//節流
ErrorSingle[1](
	bAutoStatus:=AutoStatus,
	bResetPB:=PB_Reset OR HMIPB_PB_Reset,
	bBackLS:=LS_S8_THBack,
	bOutLS:=LS_S8_THOut,
	bSOL:=SOL_S8_TH,
	bErrorStatus_Back=>Error_LS_S8_THBack,
	bErrorStatus_Out=>Error_LS_S8_THOut);
//換卡子
ErrorSingle[2](
	bAutoStatus:=AutoStatus,
	bResetPB:=PB_Reset OR HMIPB_PB_Reset,
	bBackLS:=LS_S8_FixBack,
	bOutLS:=LS_S8_FixOut,
	bSOL:=SOL_S8_Fix,
	bErrorStatus_Back=>Error_LS_S8_FixBack,
	bErrorStatus_Out=>Error_LS_S8_FixOut);
ErrorSingle[3](
	bAutoStatus:=AutoStatus,
	bResetPB:=PB_Reset OR HMIPB_PB_Reset,
	bBackLS:=LS_S8_FixMoveBack,
	bOutLS:=LS_S8_FixMoveOut,
	bSOL:=SOL_S8_FixMove,
	bErrorStatus_Back=>Error_LS_S8_FixMoveBack,
	bErrorStatus_Out=>Error_LS_S8_FixMoveOut);
ErrorSingle[4](
	bAutoStatus:=AutoStatus,
	bResetPB:=PB_Reset OR HMIPB_PB_Reset,
	bBackLS:=LS_S8_TurnBack,
	bOutLS:=LS_S8_TurnOut,
	bSOL:=SOL_S8_Turn,
	bErrorStatus_Back=>Error_LS_S8_TurnBack,
	bErrorStatus_Out=>Error_LS_S8_TurnOut);
ErrorSingle[5](
	bAutoStatus:=AutoStatus,
	bResetPB:=PB_Reset OR HMIPB_PB_Reset,
	bBackLS:=LS_S8_ClipBack,
	bOutLS:=LS_S8_ClipOut,
	bSOL:=SOL_S8_Clip,
	bErrorStatus_Back=>Error_LS_S8_ClipBack,
	bErrorStatus_Out=>Error_LS_S8_ClipOut);
//異常
ErrorStatus[8]:=
Error_LS_S8_MoveBack OR
Error_LS_S8_MoveBack OR
Error_LS_S8_UpDownBack OR
Error_LS_S8_UpDownOut OR
Error_SNR_S8_VacuumF OR
Error_SNR_S8_VacuumR OR
Error_OMRON_FQ2_Error;

ErrorStatus_TH[8]:=
Error_LS_S8_THBack OR
Error_LS_S8_THOut;

ErrorStatus_S8_Fix:=
Error_LS_S8_FixBack OR
Error_LS_S8_FixOut OR
Error_LS_S8_FixMoveBack OR
Error_LS_S8_FixMoveOut OR
Error_LS_S8_TurnBack OR
Error_LS_S8_TurnOut OR
Error_LS_S8_ClipBack OR
Error_LS_S8_ClipOut;
//RESET
IF PB_Reset OR HMIPB_PB_Reset THEN
	Error_SNR_S8_VacuumF:=FALSE;
	Error_SNR_S8_VacuumR:=FALSE;
	Error_OMRON_FQ2_Error:=FALSE;
END_IF;
END_PROGRAM

PROGRAM prError_S10
VAR
    ErrorDouble : ARRAY[0..9] of fbErrorDouble;
    ErrorSingle : ARRAY[0..9] of fbErrorSingle;
END_VAR
VAR_EXTERNAL
    AutoStatus : BOOL;
    PB_Reset : BOOL;
    HMIPB_PB_Reset : BOOL;
    LS_S10_MoveBack : BOOL;
    LS_S10_MoveOut : BOOL;
    SOL_S10_MoveBack : BOOL;
    SOL_S10_MoveOut : BOOL;
    Error_LS_S10_MoveBack : BOOL;
    Error_LS_S10_MoveOut : BOOL;
    LS_S10_UpDownBack : BOOL;
    LS_S10_UpDownOut : BOOL;
    SOL_S10_UpDown : BOOL;
    Error_LS_S10_UpDownBack : BOOL;
    Error_LS_S10_UpDownOut : BOOL;
    ErrorStatus : ARRAY[0..19] OF BOOL;
    ErrorStatus_TH : ARRAY[0..19] OF BOOL;
    LS_S10_THBack : BOOL;
    LS_S10_THOut : BOOL;
    SOL_S10_TH : BOOL;
    Error_LS_S10_THBack : BOOL;
    Error_LS_S10_THOut : BOOL;
    LS_S10_ClipFBack : BOOL;
    LS_S10_ClipFOut : BOOL;
    SOL_S10_ClipF : BOOL;
    Error_LS_S10_ClipFBack : BOOL;
    Error_LS_S10_ClipFOut : BOOL;
    LS_S10_ClipRBack : BOOL;
    LS_S10_ClipROut : BOOL;
    SOL_S10_ClipR : BOOL;
    Error_LS_S10_ClipRBack : BOOL;
    Error_LS_S10_ClipROut : BOOL;
END_VAR
//**********************************************************************************************************************
(*Station10*)
//**********************************************************************************************************************
ErrorDouble[0](
	bAutoStatus:=AutoStatus,
	bResetPB:=PB_Reset OR HMIPB_PB_Reset,
	bBackLS:=LS_S10_MoveBack,
	bOutLS:=LS_S10_MoveOut,
	bBackSOL:=SOL_S10_MoveBack,
	bOutSOL:=SOL_S10_MoveOut,
	bErrorStatus_Back=>Error_LS_S10_MoveBack,
	bErrorStatus_Out=>Error_LS_S10_MoveOut);

ErrorSingle[0](
	bAutoStatus:=AutoStatus,
	bResetPB:=PB_Reset OR HMIPB_PB_Reset,
	bBackLS:=LS_S10_UpDownBack,
	bOutLS:=LS_S10_UpDownOut,
	bSOL:=SOL_S10_UpDown,
	bErrorStatus_Back=>Error_LS_S10_UpDownBack,
	bErrorStatus_Out=>Error_LS_S10_UpDownOut);

ErrorSingle[1](
	bAutoStatus:=AutoStatus,
	bResetPB:=PB_Reset OR HMIPB_PB_Reset,
	bBackLS:=LS_S10_ClipFBack,
	bOutLS:=LS_S10_ClipFOut,
	bSOL:=SOL_S10_ClipF,
	bErrorStatus_Back=>Error_LS_S10_ClipFBack,
	bErrorStatus_Out=>Error_LS_S10_ClipFOut);

ErrorSingle[2](
	bAutoStatus:=AutoStatus,
	bResetPB:=PB_Reset OR HMIPB_PB_Reset,
	bBackLS:=LS_S10_ClipRBack,
	bOutLS:=LS_S10_ClipROut,
	bSOL:=SOL_S10_ClipR,
	bErrorStatus_Back=>Error_LS_S10_ClipRBack,
	bErrorStatus_Out=>Error_LS_S10_ClipROut);
//節流
ErrorSingle[3](
	bAutoStatus:=AutoStatus,
	bResetPB:=PB_Reset OR HMIPB_PB_Reset,
	bBackLS:=LS_S10_THBack,
	bOutLS:=LS_S10_THOut,
	bSOL:=SOL_S10_TH,
	bErrorStatus_Back=>Error_LS_S10_THBack,
	bErrorStatus_Out=>Error_LS_S10_THOut);

//異常
ErrorStatus[10]:=
Error_LS_S10_MoveBack OR
Error_LS_S10_MoveBack OR
Error_LS_S10_UpDownBack OR
Error_LS_S10_UpDownOut OR
Error_LS_S10_ClipFBack OR
Error_LS_S10_ClipFOut OR
Error_LS_S10_ClipRBack OR
Error_LS_S10_ClipROut;

ErrorStatus_TH[10]:=
Error_LS_S10_THBack OR
Error_LS_S10_THOut;
END_PROGRAM

PROGRAM prError_S11
VAR
    ErrorSingle : ARRAY[0..1] of fbErrorSingle;
END_VAR
VAR_EXTERNAL
    AutoStatus : BOOL;
    PB_Reset : BOOL;
    HMIPB_PB_Reset : BOOL;
    LS_S11_UpDownBack : BOOL;
    LS_S11_UpDownOut : BOOL;
    SOL_S11_UpDown : BOOL;
    Error_LS_S11_UpDownBack : BOOL;
    Error_LS_S11_UpDownOut : BOOL;
    ErrorStatus : ARRAY[0..19] OF BOOL;
END_VAR
//**********************************************************************************************************************
(*Station11*)
//**********************************************************************************************************************
ErrorSingle[0](
	bAutoStatus:=AutoStatus,
	bResetPB:=PB_Reset OR HMIPB_PB_Reset,
	bBackLS:=LS_S11_UpDownBack,
	bOutLS:=LS_S11_UpDownOut,
	bSOL:=SOL_S11_UpDown,
	bErrorStatus_Back=>Error_LS_S11_UpDownBack,
	bErrorStatus_Out=>Error_LS_S11_UpDownOut);

ErrorStatus[11]:=
Error_LS_S11_UpDownBack OR
Error_LS_S11_UpDownOut;
END_PROGRAM

PROGRAM prError_S13
VAR
    ErrorSingle : ARRAY[0..1] of fbErrorSingle;
END_VAR
VAR_EXTERNAL
    AutoStatus : BOOL;
    PB_Reset : BOOL;
    HMIPB_PB_Reset : BOOL;
    LS_S13_UpDownBack : BOOL;
    LS_S13_UpDownOut : BOOL;
    SOL_S13_UpDown : BOOL;
    Error_LS_S13_UpDownBack : BOOL;
    Error_LS_S13_UpDownOut : BOOL;
    ErrorStatus : ARRAY[0..19] OF BOOL;
END_VAR
//**********************************************************************************************************************
(*Station13*)
//**********************************************************************************************************************
ErrorSingle[0](
	bAutoStatus:=AutoStatus,
	bResetPB:=PB_Reset OR HMIPB_PB_Reset,
	bBackLS:=LS_S13_UpDownBack,
	bOutLS:=LS_S13_UpDownOut,
	bSOL:=SOL_S13_UpDown,
	bErrorStatus_Back=>Error_LS_S13_UpDownBack,
	bErrorStatus_Out=>Error_LS_S13_UpDownOut);

ErrorStatus[13]:=
Error_LS_S13_UpDownBack OR
Error_LS_S13_UpDownOut;
END_PROGRAM

PROGRAM prError_S15
VAR
    ErrorSingle : ARRAY[0..1] of fbErrorSingle;
END_VAR
VAR_EXTERNAL
    AutoStatus : BOOL;
    PB_Reset : BOOL;
    HMIPB_PB_Reset : BOOL;
    LS_S15_UpDownBack : BOOL;
    LS_S15_UpDownOut : BOOL;
    SOL_S15_UpDown : BOOL;
    Error_LS_S15_UpDownBack : BOOL;
    Error_LS_S15_UpDownOut : BOOL;
    ErrorStatus : ARRAY[0..19] OF BOOL;
END_VAR
//**********************************************************************************************************************
(*Station15*)
//**********************************************************************************************************************
ErrorSingle[0](
	bAutoStatus:=AutoStatus,
	bResetPB:=PB_Reset OR HMIPB_PB_Reset,
	bBackLS:=LS_S15_UpDownBack,
	bOutLS:=LS_S15_UpDownOut,
	bSOL:=SOL_S15_UpDown,
	bErrorStatus_Back=>Error_LS_S15_UpDownBack,
	bErrorStatus_Out=>Error_LS_S15_UpDownOut);

ErrorStatus[15]:=
Error_LS_S15_UpDownBack OR
Error_LS_S15_UpDownOut;
END_PROGRAM

PROGRAM prStation1
VAR
    AutoFlow : INT;
    Rtrig_test : R_TRIG;
    TON_CT : TON;
END_VAR
VAR_EXTERNAL
    IndexData : ARRAY[0..19] OF stIndexData;
    DisablePB : ARRAY[0..19] OF BOOL;
    TestPB : ARRAY[0..19] OF BOOL;
    SystemReadyStatus : BOOL;
    AutoStatus : BOOL;
    ErrorStatus : ARRAY[0..19] OF BOOL;
    Error_PB_EStop : BOOL;
    YAMAHA_Load_Start : BOOL;
    MachineRunStatus : BOOL;
    YAMAHA_Load_Finish : BOOL;
    CycleTime : ARRAY[0..19] OF REAL;
    BatchIndexCount : DINT;
    HMIPB_YAMAHA_Load_Start : BOOL;
    HMIPB_OMRON_FQ2_Trig : BOOL;
    Error_LS_Door : BOOL;
    StepMode : BOOL;
END_VAR
(*
程序名稱:第1站上料流程
作者:蔡相偉
版本,日期,版本資訊:
1.0.0		2017/11/21		初始版本
PowerOn=0
Idle=1
上料開始=2
上料完成=3
*)
//本站狀態判斷
IF IndexData[1].OKFlag[1]
	OR IndexData[1].NGFlag[1] THEN
	IndexData[1].FinishFlag[1]:=TRUE;
END_IF;
(*
//前站狀態判斷
IF NOT(IndexData[10].FinishFlag[9]
	AND IndexData[10].OKFlag[9]
	AND NOT(IndexData[10].NGFlag[9])) THEN
	IndexData[10].NGFlag[10]:=TRUE;
END_IF;
*)
//本站關閉判斷
IF DisablePB[1] AND NOT(IndexData[1].FinishFlag[1]) THEN
	IndexData[1].NGFlag[1]:=TRUE;
END_IF;
//異常放棄
IF (ErrorStatus[1] OR Error_PB_EStop) AND NOT(IndexData[1].FinishFlag[1]) THEN
	IndexData[1].NGFlag[1]:=TRUE;
END_IF;

Rtrig_test(CLK:=TestPB[1]);
//PowerOn=0
IF NOT(SystemReadyStatus AND AutoStatus AND NOT(ErrorStatus[1]) AND NOT(Error_PB_EStop)) THEN
	Autoflow:=0;
END_IF;

//Idle=1
IF AutoFlow=0 AND SystemReadyStatus AND AutoStatus AND NOT(ErrorStatus[1]) AND NOT(Error_PB_EStop) THEN
	AutoFlow:=1;
END_IF;

IF AutoFlow=3 AND NOT(YAMAHA_Load_Start) AND IndexData[1].FinishFlag[1] THEN
	AutoFlow:=1;
END_IF;

//上料開始=2
IF Autoflow=1
	AND AutoStatus
	AND NOT(DisablePB[1])
	AND (MachineRunStatus AND NOT(IndexData[1].FinishFlag[1]) OR Rtrig_test.Q) THEN
	Autoflow:=2;
END_IF;
IF AutoFlow=2 THEN
	HMIPB_YAMAHA_Load_Start:=TRUE;
END_IF;
IF YAMAHA_Load_Finish OR ErrorStatus[1] OR Error_LS_Door THEN
	HMIPB_YAMAHA_Load_Start:=FALSE;
END_IF;

//上料完成=3
IF AutoFlow=2 AND (YAMAHA_Load_Finish) THEN
	BatchIndexCount:=BatchIndexCount+1;
	AutoFlow:=3;
END_IF;
IF AutoFlow=3 THEN
	IndexData[1].OKFlag[1]:=TRUE;
END_IF;
//IndexCount
(*IF BatchIndexCount<0 THEN
	BatchIndexCount:=0;
END_IF;*)
//*************************************************************************
//Cycle Time
//*************************************************************************
TON_CT(In:=AutoFlow>1, PT:=t#500s);
IF AutoFlow>1 THEN
CycleTime[1]:=LINT_TO_REAL(TimeToNanoSec( TON_CT.ET))/1000000000.0;
END_IF;
END_PROGRAM

PROGRAM prStation1_Robot
VAR
    R_TRIG1 : R_TRIG;
    R_TRIG2 : R_TRIG;
    R_TRIG3 : R_TRIG;
END_VAR
VAR_EXTERNAL
    HMIPB_YAMAHA_Unload_OKStart : BOOL;
    YAMAHA_Unload_OKStart : BOOL;
    YAMAHA_Unload_NGStart : BOOL;
    HMIPB_YAMAHA_Unload_NGStart : BOOL;
    YAMAHA_Load_Start : BOOL;
    HMIPB_YAMAHA_Load_Start : BOOL;
    YAMAHA_UnLoad_Ready : BOOL;
    HMIPB_YAMAHA_UnLoad_Ready : BOOL;
    HMIPB_YAMAHA_Load_Ready : BOOL;
    YAMAHA_Load_Ready : BOOL;
    HMIPB_YAMAHA_Unload_ChangePanelStart : BOOL;
    YAMAHA_Unload_ChangePanelStart : BOOL;
    HMIPB_YAMAHA_Load_ChangePanelStart : BOOL;
    YAMAHA_Load_ChangePanelStart : BOOL;
    HMIPB_YAMAHA_ORG : BOOL;
    YAMAHA_ORG : BOOL;
    HMIPB_YAMAHA_S_Enable : BOOL;
    YAMAHA_S_Enable : BOOL;
    HMIPB_YAMAHA_S_Control : BOOL;
    YAMAHA_S_Control : BOOL;
    HMIPB_YAMAHA_S_Stop : BOOL;
    YAMAHA_S_Stop : BOOL;
    HMIPB_YAMAHA_S_AutoRun : BOOL;
    YAMAHA_S_AutoRun : BOOL;
    HMIPB_YAMAHA_S_INCHome : BOOL;
    YAMAHA_S_INCHome : BOOL;
    HMIPB_YAMAHA_S_ProgramReset : BOOL;
    YAMAHA_S_ProgramReset : BOOL;
    HMIPB_YAMAHA_S_AlarmReset : BOOL;
    YAMAHA_S_AlarmReset : BOOL;
    HMIPB_YAMAHA_S_ABSHome : BOOL;
    YAMAHA_S_ABSHome : BOOL;
    PB_EStop : BOOL;
    SNR_S1_Door1 : BOOL;
    SNR_S1_Door2 : BOOL;
    SNR_S1_Door3 : BOOL;
    SNR_S1_Door4 : BOOL;
    SystemReadyStatus : BOOL;
    YAMAHA_S_State_CPUOK : BOOL;
    YAMAHA_S_State_Enable : BOOL;
    Error_PB_EStop : BOOL;
    Error_LS_Door : BOOL;
    YAMAHA_S_State_Homed : BOOL;
    YAMAHA_S_State_ProgramReset : BOOL;
    YAMAHA_S_State_RobotProgramRun : BOOL;
END_VAR
//Define
YAMAHA_Unload_OKStart:=HMIPB_YAMAHA_Unload_OKStart;
YAMAHA_Unload_NGStart:=HMIPB_YAMAHA_Unload_NGStart;
YAMAHA_Load_Start:=HMIPB_YAMAHA_Load_Start;
//YAMAHA_UnLoad_Ready:=HMIPB_YAMAHA_UnLoad_Ready;
//YAMAHA_Load_Ready:=HMIPB_YAMAHA_Load_Ready;
YAMAHA_S_Control:=HMIPB_YAMAHA_S_Control;
YAMAHA_S_AutoRun:=HMIPB_YAMAHA_S_AutoRun;
YAMAHA_S_INCHome:=HMIPB_YAMAHA_S_INCHome;
YAMAHA_S_ProgramReset:=HMIPB_YAMAHA_S_ProgramReset;
YAMAHA_S_AlarmReset:=HMIPB_YAMAHA_S_AlarmReset;
YAMAHA_S_ABSHome:=HMIPB_YAMAHA_S_ABSHome;

//********************************************************************************************************
//ROBOT伺服ON流程
//********************************************************************************************************
R_TRIG1(Clk:=(SystemReadyStatus AND YAMAHA_S_State_CPUOK) OR HMIPB_YAMAHA_S_Enable);
IF R_TRIG1.Q THEN
	YAMAHA_S_Enable:=TRUE;
END_IF;
IF YAMAHA_S_State_Enable THEN
	YAMAHA_S_Enable:=FALSE;
END_IF;
//********************************************************************************************************
//STOP ON
//********************************************************************************************************
YAMAHA_S_Stop:=
HMIPB_YAMAHA_S_Stop AND
NOT(Error_PB_EStop) AND
NOT(Error_LS_Door);
//********************************************************************************************************
//程序復位和執行
//********************************************************************************************************
R_TRIG2(Clk:=YAMAHA_S_State_Homed AND YAMAHA_S_State_Enable AND YAMAHA_S_Stop AND HMIPB_YAMAHA_S_ProgramReset);
R_TRIG3(Clk:=YAMAHA_S_State_Homed AND YAMAHA_S_State_Enable AND YAMAHA_S_Stop AND YAMAHA_S_State_ProgramReset AND HMIPB_YAMAHA_S_AutoRun);
IF R_TRIG2.Q THEN
	YAMAHA_S_ProgramReset:=TRUE;
END_IF;
IF YAMAHA_S_State_ProgramReset THEN
	HMIPB_YAMAHA_S_ProgramReset:=FALSE;
END_IF;
IF R_TRIG3.Q THEN
	YAMAHA_S_AutoRun:=TRUE;
END_IF;
IF YAMAHA_S_State_RobotProgramRun AND NOT(YAMAHA_S_State_ProgramReset) THEN
	YAMAHA_S_AutoRun:=FALSE;
	HMIPB_YAMAHA_S_AutoRun:=FALSE;
END_IF;
END_PROGRAM

PROGRAM prStation1_PanelLoad
VAR
    Autoflow : INT;
    Initflow : INT;
    interlockback : ARRAY[0..2] OF BOOL;
    interlockout : ARRAY[0..2] OF BOOL;
    solStatus : ARRAY[0..2] OF BOOL;
    R_TRIG_1 : ARRAY[0..2] OF R_TRIG;
    F_TRIG_1 : F_TRIG;
    ErrorLS : BOOL;
    StartFlag : BOOL;
    TON_1 : TON;
    TON_2 : TON;
    TON_3 : TON;
    Rtrig_test : R_TRIG;
END_VAR
VAR_EXTERNAL
    HMIPB_SOL_S1_Load_PanelUpDown1Back : BOOL;
    SOL_S1_Load_PanelUpDown1Back : BOOL;
    SOL_S1_Load_PanelUpDown1Out : BOOL;
    LS_S1_Load_PanelUpDown1Back : BOOL;
    HMIPB_SOL_S1_Load_PanelUpDown1Out : BOOL;
    AutoStatus : BOOL;
    LS_S1_Load_PanelUpDown1Out : BOOL;
    HMIPB_SOL_S1_Load_PanelUpDown2Back : BOOL;
    SOL_S1_Load_PanelUpDown2Back : BOOL;
    SOL_S1_Load_PanelUpDown2Out : BOOL;
    LS_S1_Load_PanelUpDown2Back : BOOL;
    HMIPB_SOL_S1_Load_PanelUpDown2Out : BOOL;
    LS_S1_Load_PanelUpDown2Out : BOOL;
    HMIPB_SOL_S1_Load_PanelClip : BOOL;
    SOL_S1_Load_PanelClip : BOOL;
    SystemReadyStatus : BOOL;
    ErrorStatus : ARRAY[0..19] OF BOOL;
    Error_PB_EStop : BOOL;
    SNR_S1_Load_PanelFeed : BOOL;
    LS_S1_Load_PanelClip1Out : BOOL;
    LS_S1_Load_PanelClip2Out : BOOL;
    LS_S1_Load_PanelClip2Back : BOOL;
    LS_S1_Load_PanelClip1Back : BOOL;
    RY_S1_Load_VariableSpeedMotor : BOOL;
    Error_LS_S1_Load_PanelUpDown1Back : BOOL;
    Error_LS_S1_Load_PanelUpDown1Out : BOOL;
    Error_LS_S1_Load_PanelUpDown2Back : BOOL;
    Error_LS_S1_Load_PanelUpDown2Out : BOOL;
    Error_LS_S1_Load_PanelClip1Back : BOOL;
    Error_LS_S1_Load_PanelClip1Out : BOOL;
    Error_LS_S1_Load_PanelClip2Back : BOOL;
    Error_LS_S1_Load_PanelClip2Out : BOOL;
    ErrorStatus_S1_Load : BOOL;
    Error_SNR_S1_Load_PanelFeed : BOOL;
    PB_Reset : BOOL;
    HMIPB_PB_Reset : BOOL;
    StepMode : BOOL;
    Manual2AutoFlag : BOOL;
END_VAR
(*
程序名稱: Panel LOAD程序
作者:蔡相偉
版本,日期,版本資訊:
1.0.0		2017/11/16		初始版本

PowerOn=0
Idle=1
Panel出盤程序開始=10
第1段,第2段出=2
夾持出=3
第2段回=4
夾持回=5
第1段回=6
第1段到回=7
*)
//***************************************************************************************************************
//Define
ErrorLS:=ErrorStatus_S1_Load;
StartFlag:=TON_1.Q;
TON_1(In:=NOT(SNR_S1_Load_PanelFeed) AND NOT(RY_S1_Load_VariableSpeedMotor), PT:=t#5s);
//PowerOn=0
IF NOT(SystemReadyStatus AND NOT(ErrorLS) AND  NOT(Error_PB_Estop) AND AutoStatus) THEN
	Autoflow:=0;
END_IF;

//Idle=1
IF AutoFlow=0 AND SystemReadyStatus AND NOT(ErrorLS) AND  NOT(Error_PB_Estop) AND AutoStatus THEN
	AutoFlow:=1;
END_IF;

IF Autoflow=7 AND (Error_SNR_S1_Load_PanelFeed OR SNR_S1_Load_PanelFeed) THEN
	Autoflow:=1;
END_IF;

//第1段,第2段出=2
IF Autoflow=1 AND NOT(Error_SNR_S1_Load_PanelFeed) AND StartFlag THEN
	Autoflow:=2;
END_IF;

//承盤夾持出=3
IF Autoflow=2 AND LS_S1_Load_PanelUpDown1Out AND LS_S1_Load_PanelUpDown2Out AND (Rtrig_test.Q OR NOT(StepMode)) THEN
	Autoflow:=3;
END_IF;
TON_2(In:= Autoflow=3 AND LS_S1_Load_PanelClip1Out AND LS_S1_Load_PanelClip2Out , PT:=t#300ms);

//第2段回=4
IF Autoflow=3 AND TON_2.Q AND (Rtrig_test.Q OR NOT(StepMode)) THEN
	Autoflow:=4;
END_IF;
TON_3(In:=Autoflow=4 AND LS_S1_Load_PanelUpDown2Back, PT:=t#300ms);

//承盤夾持回=5
IF Autoflow=4 AND TON_3.Q AND (Rtrig_test.Q OR NOT(StepMode)) THEN
	Autoflow:=5;
END_IF;

//第1段回=6
IF Autoflow=5 AND  LS_S1_Load_PanelClip1Back AND LS_S1_Load_PanelClip2Back AND (Rtrig_test.Q OR NOT(StepMode)) THEN
	Autoflow:=6;
END_IF;

//第1段到回=7
IF Autoflow=6 AND  LS_S1_Load_PanelUpDown1Back AND (Rtrig_test.Q OR NOT(StepMode)) THEN
	Autoflow:=7;
END_IF;
IF Autoflow=7 AND NOT(SNR_S1_Load_PanelFeed) THEN
	Error_SNR_S1_Load_PanelFeed:=TRUE;
END_IF;

//***************************************************************************************************************
//下夾板出盤下降第1段回電磁閥
interlockback[0]:=TRUE;
IF ((HMIPB_SOL_S1_Load_PanelUpDown1Back AND NOT(AutoStatus)) OR Autoflow=6 OR Initflow=3) AND interlockback[0] THEN
	SOL_S1_Load_PanelUpDown1Back:=TRUE;
	SOL_S1_Load_PanelUpDown1Out:=FALSE;
END_IF;
IF LS_S1_Load_PanelUpDown1Back THEN
	SOL_S1_Load_PanelUpDown1Back:=FALSE;
END_IF;

//下夾板出盤下降第1段出電磁閥
interlockout[0]:=TRUE;
IF ((HMIPB_SOL_S1_Load_PanelUpDown1Out AND NOT(AutoStatus)) OR Autoflow=2) AND interlockout[0] THEN
	SOL_S1_Load_PanelUpDown1Back:=FALSE;
	SOL_S1_Load_PanelUpDown1Out:=TRUE;
END_IF;
IF LS_S1_Load_PanelUpDown1Out THEN
	SOL_S1_Load_PanelUpDown1Out:=FALSE;
END_IF;
//***************************************************************************************************************
//下夾板出盤下降第2段回電磁閥
interlockback[1]:=TRUE;
IF ((HMIPB_SOL_S1_Load_PanelUpDown2Back AND NOT(AutoStatus)) OR Autoflow=4 OR Initflow=3) AND interlockback[1] THEN
	SOL_S1_Load_PanelUpDown2Back:=TRUE;
	SOL_S1_Load_PanelUpDown2Out:=FALSE;
END_IF;
IF LS_S1_Load_PanelUpDown2Back THEN
	SOL_S1_Load_PanelUpDown2Back:=FALSE;
END_IF;

//下夾板出盤下降第2段出電磁閥
interlockout[1]:=LS_S1_Load_PanelUpDown1Out AND NOT(SNR_S1_Load_PanelFeed);
IF ((HMIPB_SOL_S1_Load_PanelUpDown2Out AND NOT(AutoStatus)) OR Autoflow=2) AND interlockout[1] THEN
	SOL_S1_Load_PanelUpDown2Back:=FALSE;
	SOL_S1_Load_PanelUpDown2Out:=TRUE;
END_IF;
IF LS_S1_Load_PanelUpDown2Out THEN
	SOL_S1_Load_PanelUpDown2Out:=FALSE;
END_IF;
//***************************************************************************************************************
(*下夾板出盤承載電磁閥*)
R_TRIG_1[2](CLK:=HMIPB_SOL_S1_Load_PanelClip AND NOT(AutoStatus));
interlockback[2]:=TRUE;
interlockout[2]:=LS_S1_Load_PanelUpDown1Out;
(*SET*)
IF ((R_TRIG_1[2].Q AND NOT(solStatus[2])) OR Autoflow=3) AND interlockout[2] THEN
	SOL_S1_Load_PanelClip:=TRUE;
END_IF;
(*RESET*)
IF ((R_TRIG_1[2].Q AND (solStatus[2])) OR Autoflow=5 OR Initflow=2) AND interlockback[2] THEN
	SOL_S1_Load_PanelClip:=FALSE;
END_IF;
(*STATUS*)
solStatus[2]:=SOL_S1_Load_PanelClip;

//***************************************************************************************************************
(*
程序名稱: Panel LOAD RESET程序
作者:蔡相偉
版本,日期,版本資訊:
1.0.0		2017/11/16		初始版本

PowerOn=0
Idle=1
夾持回=2
第1段回,第2段回=3
*)
//***************************************************************************************************************
//PowerOn=0
IF NOT(SystemReadyStatus) THEN
	Initflow:=0;
END_IF;

//Idle=1
IF Initflow=0 AND SystemReadyStatus THEN
	Initflow:=1;
END_IF;

IF Initflow=3 AND LS_S1_Load_PanelUpDown1Back AND LS_S1_Load_PanelUpDown2Back THEN
	Initflow:=1;
END_IF;

F_TRIG_1(Clk:=ErrorLS OR Error_PB_Estop);
//夾持回=2
IF Initflow=1 AND (F_TRIG_1.Q OR Manual2AutoFlag) THEN
	Initflow:=2;
END_IF;

//第1段回,第2段回=3
IF Initflow=2 AND LS_S1_Load_PanelClip1Back AND LS_S1_Load_PanelClip2Back THEN
	Initflow:=3;
END_IF;
END_PROGRAM

PROGRAM prStation1_FeedPanelLoad
VAR
    Autoflow : INT;
    interlockback : ARRAY[0..3] OF BOOL;
    interlockout : ARRAY[0..3] OF BOOL;
    solStatus : ARRAY[0..3] OF BOOL;
    R_TRIG_1 : ARRAY[0..3] OF R_TRIG;
    ErrorLS : BOOL;
    StartFlag : BOOL;
    TON_1 : TON;
    TON_2 : TON;
    TON_3 : TON;
    TON_4 : TON;
    TON_5 : TON;
    TON_6 : TON;
    F_TRIG_1 : F_TRIG;
    centermotorStartflag : BOOL;
    Rtrig_test : R_TRIG;
    Initflow : INT;
END_VAR
VAR_EXTERNAL
    HMIPB_SOL_S1_Load_PanelUpDown1Back : BOOL;
    SOL_S1_Load_PanelUpDown1Back : BOOL;
    SOL_S1_Load_PanelUpDown1Out : BOOL;
    LS_S1_Load_PanelUpDown1Back : BOOL;
    HMIPB_SOL_S1_Load_PanelUpDown1Out : BOOL;
    AutoStatus : BOOL;
    LS_S1_Load_PanelUpDown1Out : BOOL;
    HMIPB_SOL_S1_Load_PanelUpDown2Back : BOOL;
    SOL_S1_Load_PanelUpDown2Back : BOOL;
    SOL_S1_Load_PanelUpDown2Out : BOOL;
    LS_S1_Load_PanelUpDown2Back : BOOL;
    HMIPB_SOL_S1_Load_PanelUpDown2Out : BOOL;
    LS_S1_Load_PanelUpDown2Out : BOOL;
    HMIPB_SOL_S1_Load_PanelClip : BOOL;
    SOL_S1_Load_PanelClip : BOOL;
    HMIPB_SOL_S1_Load_FixClip : BOOL;
    SOL_S1_Load_FixClip : BOOL;
    HMIPB_SOL_S1_Load_ConveyorClip : BOOL;
    SOL_S1_Load_ConveyorClip : BOOL;
    HMIPB_SOL_S1_Load_UpDown : BOOL;
    SOL_S1_Load_UpDown : BOOL;
    HMIPB_RY_S1_Load_VariableSpeedMotor : BOOL;
    RY_S1_Load_VariableSpeedMotor : BOOL;
    RY_S1_Load_FixSpeedMotor : BOOL;
    HMIPB_RY_S1_Load_FixSpeedMotor : BOOL;
    SNR_S1_Load_PanelFeed : BOOL;
    SNR_S1_Load_PanelClip : BOOL;
    SystemReadyStatus : BOOL;
    ErrorStatus : ARRAY[0..19] OF BOOL;
    ErrorStatus_TH : ARRAY[0..19] OF BOOL;
    RY_S1_Center_VariableSpeedMotor : BOOL;
    HMIPB_RY_S1_Center_VariableSpeedMotor : BOOL;
    Error_PB_EStop : BOOL;
    ErrorStatus_S1_FeedPanelLoad : BOOL;
    HMIPB_SOL_S1_Load_AlignmentClip : BOOL;
    SOL_S1_Load_AlignmentClip : BOOL;
    YAMAHA_Load_ChangePanelStart : BOOL;
    HMIPB_YAMAHA_Load_ChangePanelStart : BOOL;
    SNR_AirSource : BOOL;
    SNR_S1_Load_Feed : BOOL;
    SNR_S1_UnLoad_Feed : BOOL;
    LS_S1_Load_FixClipOut : BOOL;
    LS_S1_Load_AlignmentClipOut : BOOL;
    HMIPB_YAMAHA_Unload_ChangePanelStart : BOOL;
    LS_S1_Load_UpDownOut : BOOL;
    LS_S1_Load_ConveyorClip1Out : BOOL;
    LS_S1_Load_ConveyorClip2Out : BOOL;
    LS_S10_ClipFBack : BOOL;
    LS_S1_Load_UpDownBack : BOOL;
    LS_S1_Load_ConveyorClip1Back : BOOL;
    LS_S1_Load_ConveyorClip2Back : BOOL;
    LS_S1_Load_FixClipBack : BOOL;
    LS_S1_Load_AlignmentClipBack : BOOL;
    YAMAHA_Load_Ready : BOOL;
    YAMAHA_Load_Finish : BOOL;
    YAMAHA_Load_Start : BOOL;
    YAMAHA_Unload_ChangePanelStart : BOOL;
    LS_S1_UnLoad_UpDownBack : BOOL;
    SOL_S1_UnLoad_UpDown : BOOL;
    StepMode : BOOL;
    LS_S1_UnLoad_PanelUpDown1Back : BOOL;
    LS_S1_UnLoad_PanelUpDown2Back : BOOL;
    Manual2AutoFlag : BOOL;
    LS_S1_UnLoad_PanelClip1Back : BOOL;
    LS_S1_UnLoad_PanelClip2Back : BOOL;
END_VAR
(*
程序名稱: 出盤程序
作者:蔡相偉
版本,日期,版本資訊:
1.0.0		2017/11/16		初始版本

PowerOn=0--->
Idle=1--->
換盤程序開始=2|--->工件取放處有盤=10--->固定,活動夾持出=11--->上下出=12--->軌道夾持出=13--->上下回=14--->軌道夾持回=15--->20
						  |--->工件取放處無盤=20--->軌道夾持回=21--->固定,活動夾持出=22--->馬達ON=23--->馬達運行中=24--->盤到位,馬達停止=25--->固定邊夾持回=26--->活動邊夾持回=27--->換盤完成=28--->1
*)
(*
Error Code
1:緊急停止
2:磁簧異常
*)
//***************************************************************************************************************
//Define
ErrorLS:=
ErrorStatus_S1_FeedPanelLoad;
//***************************************************************************************************************
//PowerOn=0
IF NOT(SystemReadyStatus AND NOT(ErrorLS) AND  NOT(Error_PB_Estop)) THEN
	Autoflow:=0;
END_IF;

//Idle=1
IF Autoflow=0 AND SystemReadyStatus AND NOT(ErrorLS) AND  NOT(Error_PB_Estop) THEN
	Autoflow:=1;
END_IF;

IF Autoflow=28 AND NOT(YAMAHA_Load_ChangePanelStart) AND NOT(HMIPB_YAMAHA_Load_ChangePanelStart) THEN
	Autoflow:=1;
END_IF;

TON_1(In:=Autoflow=1 AND NOT(SNR_S1_Load_PanelClip), PT:=t#1s);

IF Autoflow=1 AND TON_5.Q THEN		(*READY訊號*)
	YAMAHA_Load_Ready:=TRUE;
ELSE
	YAMAHA_Load_Ready:=FALSE;
END_IF;

//換盤程序開始=2
IF Autoflow=1 AND (YAMAHA_Load_ChangePanelStart OR HMIPB_YAMAHA_Load_ChangePanelStart OR TON_1.Q) AND SNR_S1_Load_PanelFeed THEN
	Autoflow:=2;
END_IF;

//工件取放處有盤=10
IF Autoflow=2 AND SNR_S1_Load_PanelClip THEN
	Autoflow:=10;
END_IF;

//固定,活動夾持出=11
IF Autoflow=10 THEN
	Autoflow:=11;
END_IF;
IF Autoflow=11 AND SNR_S1_Load_Feed THEN
	HMIPB_YAMAHA_Unload_ChangePanelStart:=TRUE;
END_IF;
TON_4(In:=Autoflow=11 AND NOT(SNR_S1_Load_Feed), PT:=t#1s);

//上下出=12
IF Autoflow=11 AND LS_S1_Load_FixClipOut AND LS_S1_Load_AlignmentClipOut AND TON_4.Q AND (Rtrig_test.Q OR NOT(StepMode)) THEN
	Autoflow:=12;
	HMIPB_YAMAHA_Unload_ChangePanelStart:=FALSE;
END_IF;

//軌道夾持出=13
IF Autoflow=12 AND LS_S1_Load_UpDownOut AND (Rtrig_test.Q OR NOT(StepMode)) THEN
	Autoflow:=13;
END_IF;

//上下回=14
IF Autoflow=13 AND LS_S1_Load_ConveyorClip1Out AND LS_S1_Load_ConveyorClip2Out AND (Rtrig_test.Q OR NOT(StepMode)) THEN
	Autoflow:=14;
END_IF;

//軌道夾持回=15
IF Autoflow=14 AND LS_S1_Load_UpDownBack AND (Rtrig_test.Q OR NOT(StepMode)) THEN
	Autoflow:=15;
END_IF;
//***************************************************************************************************************
//工件取放處無盤=20
IF Autoflow=2 AND NOT(SNR_S1_Load_PanelClip) THEN
	Autoflow:=20;
END_IF;

IF Autoflow=15 AND LS_S1_Load_ConveyorClip1Back AND LS_S1_Load_ConveyorClip2Back THEN
	Autoflow:=20;
END_IF;

//軌道夾持回=21
IF Autoflow=20 THEN
	Autoflow:=21;
END_IF;

//固定,活動夾持出=22
IF Autoflow=21 AND LS_S1_Load_ConveyorClip1Back AND LS_S1_Load_ConveyorClip2Back AND (Rtrig_test.Q OR NOT(StepMode)) THEN
	Autoflow:=22;
END_IF;

//馬達ON=23
IF Autoflow=22 AND LS_S1_Load_FixClipOut AND LS_S1_Load_AlignmentClipOut AND SNR_S1_Load_PanelFeed THEN
	Autoflow:=23;
END_IF;
IF Autoflow=23 THEN
	HMIPB_RY_S1_Load_FixSpeedMotor:=TRUE;
	HMIPB_RY_S1_Load_VariableSpeedMotor:=TRUE;
END_IF;

//馬達運行中=24
IF Autoflow=23 AND RY_S1_Load_FixSpeedMotor AND RY_S1_Load_VariableSpeedMotor THEN
	Autoflow:=24;
END_IF;


//盤到位,馬達停止=25
IF Autoflow=24 AND TON_5.Q THEN
	Autoflow:=25;
END_IF;


//固定邊夾持回=26
IF Autoflow=25 AND NOT(RY_S1_Load_FixSpeedMotor) AND (Rtrig_test.Q OR NOT(StepMode)) THEN
	Autoflow:=26;
END_IF;

//活動邊夾持回=27
IF Autoflow=26 AND LS_S1_Load_FixClipBack AND (Rtrig_test.Q OR NOT(StepMode)) THEN
	Autoflow:=27;
END_IF;
//換盤完成=28
IF Autoflow=27 AND LS_S1_Load_AlignmentClipBack THEN
	Autoflow:=28;
END_IF;

//***************************************************************************************************************
//下夾板出盤固定邊定位電磁閥
R_TRIG_1[0](CLK:=HMIPB_SOL_S1_Load_FixClip AND NOT(AutoStatus));
interlockback[0]:=TRUE;
interlockout[0]:=TRUE;
//SET
IF ((R_TRIG_1[0].Q AND NOT(solStatus[0])) OR Autoflow=11 OR Autoflow=22) AND interlockout[0] THEN
	SOL_S1_Load_FixClip:=TRUE;
END_IF;
//RESET
IF ((R_TRIG_1[0].Q AND (solStatus[0])) OR Autoflow=26 OR Initflow=26) AND interlockback[0] THEN
	SOL_S1_Load_FixClip:=FALSE;
END_IF;
//STATUS
solStatus[0]:=SOL_S1_Load_FixClip;
//***************************************************************************************************************
//下夾板出盤活動邊定位電磁閥
R_TRIG_1[1](CLK:=HMIPB_SOL_S1_Load_AlignmentClip AND NOT(AutoStatus));
interlockback[1]:=TRUE;
interlockout[1]:=TRUE;
//SET
IF ((R_TRIG_1[1].Q AND NOT(solStatus[1])) OR Autoflow=11 OR Autoflow=22) AND interlockout[1] THEN
	SOL_S1_Load_AlignmentClip:=TRUE;
END_IF;
//RESET
IF ((R_TRIG_1[1].Q AND (solStatus[1])) OR Autoflow=27 OR Initflow=27) AND interlockback[1] THEN
	SOL_S1_Load_AlignmentClip:=FALSE;
END_IF;
//STATUS
solStatus[1]:=SOL_S1_Load_AlignmentClip;
//***************************************************************************************************************
//下夾板出盤軌道開合電磁閥
R_TRIG_1[2](CLK:=HMIPB_SOL_S1_Load_ConveyorClip AND NOT(AutoStatus));
interlockback[2]:=TRUE;
interlockout[2]:=LS_S1_Load_UpDownOut AND SOL_S1_Load_UpDown;
//SET
IF ((R_TRIG_1[2].Q AND NOT(solStatus[2])) OR Autoflow=13) AND interlockout[2] THEN
	SOL_S1_Load_ConveyorClip:=TRUE;
END_IF;
//RESET
IF ((R_TRIG_1[2].Q AND (solStatus[2])) OR Autoflow=15 OR Autoflow=21 OR Initflow=21) AND interlockback[2] THEN
	SOL_S1_Load_ConveyorClip:=FALSE;
END_IF;
//STATUS
solStatus[2]:=SOL_S1_Load_ConveyorClip;
//***************************************************************************************************************
//下夾板出盤升降電磁閥
R_TRIG_1[3](CLK:=HMIPB_SOL_S1_Load_UpDown AND NOT(AutoStatus));
interlockback[3]:=TRUE;
interlockout[3]:=LS_S1_Load_AlignmentClipOut AND SOL_S1_Load_AlignmentClip AND LS_S1_Load_FixClipOut AND SOL_S1_Load_FixClip;
//RESET
IF ((R_TRIG_1[3].Q AND NOT(solStatus[3])) OR Autoflow=12) AND interlockout[3] THEN
	SOL_S1_Load_UpDown:=TRUE;
END_IF;
//RESET
IF ((R_TRIG_1[3].Q AND (solStatus[3])) OR Autoflow=14 OR Initflow=14) AND interlockback[3] THEN
	SOL_S1_Load_UpDown:=FALSE;
END_IF;
//STATUS
solStatus[3]:=SOL_S1_Load_UpDown;
//***************************************************************************************************************
//下夾板出盤調速馬達繼電器
//RESET
TON_6(In:=NOT(SNR_S1_Load_PanelFeed) AND LS_S1_Load_PanelUpDown1Back AND LS_S1_Load_PanelUpDown2Back, PT:=t#1s);
IF TON_6.Q THEN
	HMIPB_RY_S1_Load_VariableSpeedMotor:=FALSE;
END_IF;
//OUT
RY_S1_Load_VariableSpeedMotor:=HMIPB_RY_S1_Load_VariableSpeedMotor AND NOT(StepMode);
//***************************************************************************************************************
//下夾板出盤定速馬達繼電器
//RESET
TON_5(In:=SNR_S1_Load_PanelClip, PT:=t#1s);
IF TON_5.Q THEN
	HMIPB_RY_S1_Load_FixSpeedMotor:=FALSE;
END_IF;
//OUT
RY_S1_Load_FixSpeedMotor:=HMIPB_RY_S1_Load_FixSpeedMotor AND NOT(StepMode);
//***************************************************************************************************************
//下夾板下移載調速馬達繼電器
TON_2(In:=SNR_S1_Load_Feed, PT:=t#1s);
TON_3(In:=SNR_S1_UnLoad_Feed, PT:=t#1s);
IF TON_2.Q THEN
	centermotorStartflag:=TRUE;
END_IF;
IF TON_3.Q THEN
	centermotorStartflag:=FALSE;
	HMIPB_RY_S1_Center_VariableSpeedMotor:=FALSE;
END_IF;
//OUT
RY_S1_Center_VariableSpeedMotor:=
(centermotorStartflag OR
HMIPB_RY_S1_Center_VariableSpeedMotor) AND
NOT(HMIPB_YAMAHA_Load_ChangePanelStart) AND
LS_S1_Load_UpDownBack AND
NOT(SOL_S1_Load_UpDown) AND
LS_S1_UnLoad_UpDownBack AND
NOT(SOL_S1_UnLoad_UpDown) AND
NOT(StepMode);

//***************************************************************************************************************
(*
程序名稱: Feed Panel LOAD RESET程序
作者:蔡相偉
版本,日期,版本資訊:
1.0.0		2017/11/16		初始版本

PowerOn=0
Idle=1
上下回=14
軌道夾持回=21
固定邊夾持回=26
活動邊夾持回=27
*)
//***************************************************************************************************************
//PowerOn=0
IF NOT(SystemReadyStatus) THEN
	Initflow:=0;
END_IF;

//Idle=1
IF Initflow=0 AND SystemReadyStatus THEN
	Initflow:=1;
END_IF;

IF Initflow=27 AND LS_S1_Load_AlignmentClipBack THEN
	Initflow:=1;
END_IF;

F_TRIG_1(Clk:=ErrorLS OR Error_PB_Estop);
//上下回=14
IF Initflow=1 AND (F_TRIG_1.Q OR Manual2AutoFlag) THEN
	Initflow:=14;
END_IF;

//軌道夾持回=21
IF Initflow=14 AND LS_S1_Load_UpDownBack THEN
	Initflow:=21;
END_IF;

//固定邊夾持回=26
IF Initflow=21 AND LS_S1_Load_ConveyorClip1Back AND LS_S1_Load_ConveyorClip2Back THEN
	Initflow:=26;
END_IF;

//活動邊夾持回=27
IF Initflow=26 AND LS_S1_Load_FixClipBack THEN
	Initflow:=27;
END_IF;
END_PROGRAM

PROGRAM prStation1_PanelUnLoad
VAR
    Autoflow : INT;
    Initflow : INT;
    interlockback : ARRAY[0..2] OF BOOL;
    interlockout : ARRAY[0..2] OF BOOL;
    solStatus : ARRAY[0..2] OF BOOL;
    R_TRIG_1 : ARRAY[0..2] OF R_TRIG;
    F_TRIG_1 : F_TRIG;
    ErrorLS : BOOL;
    StartFlag : BOOL;
    TON_1 : TON;
    Rtrig_test : R_TRIG;
END_VAR
VAR_EXTERNAL
    RY_S1_UnLoad_VariableSpeedMotor : BOOL;
    HMIPB_SOL_S1_UnLoad_PanelUpDown1Back : BOOL;
    AutoStatus : BOOL;
    SOL_S1_UnLoad_PanelUpDown1Back : BOOL;
    SOL_S1_UnLoad_PanelUpDown1Out : BOOL;
    LS_S1_UnLoad_PanelUpDown1Back : BOOL;
    HMIPB_SOL_S1_UnLoad_PanelUpDown1Out : BOOL;
    LS_S1_UnLoad_PanelUpDown1Out : BOOL;
    HMIPB_SOL_S1_UnLoad_PanelUpDown2Back : BOOL;
    SOL_S1_UnLoad_PanelUpDown2Back : BOOL;
    SOL_S1_UnLoad_PanelUpDown2Out : BOOL;
    LS_S1_UnLoad_PanelUpDown2Back : BOOL;
    HMIPB_SOL_S1_UnLoad_PanelUpDown2Out : BOOL;
    LS_S1_UnLoad_PanelUpDown2Out : BOOL;
    HMIPB_SOL_S1_UnLoad_PanelClip : BOOL;
    SOL_S1_UnLoad_PanelClip : BOOL;
    ErrorStatus_S1_UnLoad : BOOL;
    SNR_S1_UnLoad_PanelFeed : BOOL;
    SystemReadyStatus : BOOL;
    Error_PB_EStop : BOOL;
    LS_S1_UnLoad_PanelClip1Out : BOOL;
    LS_S1_UnLoad_PanelClip2Out : BOOL;
    LS_S1_UnLoad_PanelClip1Back : BOOL;
    LS_S1_UnLoad_PanelClip2Back : BOOL;
    StepMode : BOOL;
    LS_S1_Load_PanelUpDown1Back : BOOL;
    LS_S1_Load_PanelUpDown2Back : BOOL;
    LS_S1_Load_PanelClip1Back : BOOL;
    LS_S1_Load_PanelClip2Back : BOOL;
    Manual2AutoFlag : BOOL;
END_VAR
(*
程序名稱: Panel UNLOAD程序
作者:蔡相偉
版本,日期,版本資訊:
1.0.0		2017/11/16		初始版本

PowerOn=0
Idle=1
Panel出盤程序開始=10
第1段出=2
夾持出=3
第2段出=4
夾持回=5
第1段,第2段回=6
*)
//***************************************************************************************************************
//Define
ErrorLS:=ErrorStatus_S1_UnLoad;
StartFlag:=TON_1.Q;
TON_1(In:=(SNR_S1_UnLoad_PanelFeed) AND NOT(RY_S1_UnLoad_VariableSpeedMotor), PT:=t#5s);
//PowerOn=0
IF NOT(SystemReadyStatus AND NOT(ErrorLS) AND  NOT(Error_PB_EStop) AND AutoStatus) THEN
	Autoflow:=0;
END_IF;

//Idle=1
IF AutoFlow=0 AND SystemReadyStatus AND NOT(ErrorLS) AND  NOT(Error_PB_Estop) AND AutoStatus THEN
	AutoFlow:=1;
END_IF;

IF Autoflow=6 AND LS_S1_UnLoad_PanelUpDown1Back AND LS_S1_UnLoad_PanelUpDown2Back THEN
	Autoflow:=1;
END_IF;

//第1段出=2
IF Autoflow=1 AND StartFlag THEN
	Autoflow:=2;
END_IF;

//承盤夾持出=3
IF Autoflow=2 AND LS_S1_UnLoad_PanelUpDown1Out AND (Rtrig_test.Q OR NOT(StepMode)) THEN
	Autoflow:=3;
END_IF;

//第2段出=4
IF Autoflow=3 AND LS_S1_UnLoad_PanelClip1Out AND LS_S1_UnLoad_PanelClip2Out AND (Rtrig_test.Q OR NOT(StepMode)) THEN
	Autoflow:=4;
END_IF;

//承盤夾持回=5
IF Autoflow=4 AND LS_S1_UnLoad_PanelUpDown2Out AND (Rtrig_test.Q OR NOT(StepMode)) THEN
	Autoflow:=5;
END_IF;

//第1段,第2段回=6
IF Autoflow=5 AND  LS_S1_UnLoad_PanelClip1Back AND LS_S1_UnLoad_PanelClip2Back AND (Rtrig_test.Q OR NOT(StepMode)) THEN
	Autoflow:=6;
END_IF;

//***************************************************************************************************************
//下夾板出盤下降第1段回電磁閥
interlockback[0]:=TRUE;
IF ((HMIPB_SOL_S1_UnLoad_PanelUpDown1Back AND NOT(AutoStatus)) OR Autoflow=6 OR Initflow=3) AND interlockback[0] THEN
	SOL_S1_UnLoad_PanelUpDown1Back:=TRUE;
	SOL_S1_UnLoad_PanelUpDown1Out:=FALSE;
END_IF;
IF LS_S1_UnLoad_PanelUpDown1Back THEN
	SOL_S1_UnLoad_PanelUpDown1Back:=FALSE;
END_IF;

//下夾板出盤下降第1段出電磁閥
interlockout[0]:=TRUE;
IF ((HMIPB_SOL_S1_UnLoad_PanelUpDown1Out AND NOT(AutoStatus)) OR Autoflow=2) AND interlockout[0] THEN
	SOL_S1_UnLoad_PanelUpDown1Back:=FALSE;
	SOL_S1_UnLoad_PanelUpDown1Out:=TRUE;
END_IF;
IF LS_S1_UnLoad_PanelUpDown1Out THEN
	SOL_S1_UnLoad_PanelUpDown1Out:=FALSE;
END_IF;
//***************************************************************************************************************
//下夾板出盤下降第2段回電磁閥
interlockback[1]:=TRUE;
IF ((HMIPB_SOL_S1_UnLoad_PanelUpDown2Back AND NOT(AutoStatus)) OR Autoflow=6 OR Initflow=3) AND interlockback[1] THEN
	SOL_S1_UnLoad_PanelUpDown2Back:=TRUE;
	SOL_S1_UnLoad_PanelUpDown2Out:=FALSE;
END_IF;
IF LS_S1_UnLoad_PanelUpDown2Back THEN
	SOL_S1_UnLoad_PanelUpDown2Back:=FALSE;
END_IF;

//下夾板出盤下降第2段出電磁閥
interlockout[1]:=LS_S1_UnLoad_PanelClip1Out AND LS_S1_UnLoad_PanelClip2Out AND SOL_S1_UnLoad_PanelClip;
IF ((HMIPB_SOL_S1_UnLoad_PanelUpDown2Out AND NOT(AutoStatus)) OR Autoflow=4) AND interlockout[1] THEN
	SOL_S1_UnLoad_PanelUpDown2Back:=FALSE;
	SOL_S1_UnLoad_PanelUpDown2Out:=TRUE;
END_IF;
IF LS_S1_UnLoad_PanelUpDown2Out THEN
	SOL_S1_UnLoad_PanelUpDown2Out:=FALSE;
END_IF;
//***************************************************************************************************************
(*下夾板出盤承載電磁閥*)
R_TRIG_1[2](CLK:=HMIPB_SOL_S1_UnLoad_PanelClip AND NOT(AutoStatus));
interlockback[2]:=TRUE;
interlockout[2]:=LS_S1_UnLoad_PanelUpDown1Out;
(*SET*)
IF ((R_TRIG_1[2].Q AND NOT(solStatus[2])) OR Autoflow=3) AND interlockout[2] THEN
	SOL_S1_UnLoad_PanelClip:=TRUE;
END_IF;
(*RESET*)
IF ((R_TRIG_1[2].Q AND (solStatus[2])) OR Autoflow=5 OR Initflow=2) AND interlockback[2] THEN
	SOL_S1_UnLoad_PanelClip:=FALSE;
END_IF;
(*STATUS*)
solStatus[2]:=SOL_S1_UnLoad_PanelClip;

//***************************************************************************************************************
(*
程序名稱: Panel UNLOAD RESET程序
作者:蔡相偉
版本,日期,版本資訊:
1.0.0		2017/11/16		初始版本

PowerOn=0
Idle=1
夾持回=2
第1段回,第2段回=3
*)
//***************************************************************************************************************
//PowerOn=0
IF NOT(SystemReadyStatus) THEN
	Initflow:=0;
END_IF;

//Idle=1
IF Initflow=0 AND SystemReadyStatus THEN
	Initflow:=1;
END_IF;

IF Initflow=3 AND LS_S1_UnLoad_PanelUpDown1Back AND LS_S1_UnLoad_PanelUpDown2Back THEN
	Initflow:=1;
END_IF;

F_TRIG_1(Clk:=ErrorLS OR Error_PB_Estop);
//夾持回=2
IF Initflow=1 AND (F_TRIG_1.Q OR Manual2AutoFlag) THEN
	Initflow:=2;
END_IF;

//第1段回,第2段回=3
IF Initflow=2 AND LS_S1_UnLoad_PanelClip1Back AND LS_S1_UnLoad_PanelClip2Back THEN
	Initflow:=3;
END_IF;
END_PROGRAM

PROGRAM prStation1_FeedPanelUnLoad
VAR
    Autoflow : INT;
    interlockback : ARRAY[0..3] OF BOOL;
    interlockout : ARRAY[0..3] OF BOOL;
    solStatus : ARRAY[0..3] OF BOOL;
    R_TRIG_1 : ARRAY[0..3] OF R_TRIG;
    ErrorLS : BOOL;
    StartFlag : BOOL;
    TON_1 : TON;
    TON_2 : TON;
    TON_3 : TON;
    TON_4 : TON;
    TON_5 : TON;
    TON_6 : TON;
    TON_7 : TON;
    TON_8 : TON;
    F_TRIG_1 : F_TRIG;
    TON_9 : TON;
    Rtrig_test : R_TRIG;
    Initflow : INT;
END_VAR
VAR_EXTERNAL
    HMIPB_SOL_S1_UnLoad_FixClip : BOOL;
    SOL_S1_UnLoad_FixClip : BOOL;
    AutoStatus : BOOL;
    HMIPB_SOL_S1_UnLoad_AlignmentClip : BOOL;
    SOL_S1_UnLoad_AlignmentClip : BOOL;
    HMIPB_SOL_S1_UnLoad_ConveyorClip : BOOL;
    SOL_S1_UnLoad_ConveyorClip : BOOL;
    HMIPB_SOL_S1_UnLoad_UpDown : BOOL;
    SOL_S1_UnLoad_UpDown : BOOL;
    SNR_S1_UnLoad_PanelFeed : BOOL;
    HMIPB_RY_S1_UnLoad_VariableSpeedMotor : BOOL;
    RY_S1_UnLoad_VariableSpeedMotor : BOOL;
    SNR_S1_UnLoad_PanelClip : BOOL;
    HMIPB_RY_S1_UnLoad_FixSpeedMotor : BOOL;
    RY_S1_UnLoad_FixSpeedMotor : BOOL;
    ErrorStatus_S1_FeedPanelUnLoad : BOOL;
    SystemReadyStatus : BOOL;
    Error_PB_EStop : BOOL;
    YAMAHA_Unload_ChangePanelStart : BOOL;
    HMIPB_YAMAHA_Unload_ChangePanelStart : BOOL;
    YAMAHA_Load_Ready : BOOL;
    YAMAHA_UnLoad_Ready : BOOL;
    LS_S1_UnLoad_AlignmentClipBack : BOOL;
    YAMAHA_Unload_OKStart : BOOL;
    LS_S1_UnLoad_FixClipOut : BOOL;
    LS_S1_UnLoad_AlignmentClipOut : BOOL;
    LS_S1_UnLoad_ConveyorClip1Out : BOOL;
    LS_S1_UnLoad_ConveyorClip2Out : BOOL;
    SNR_S1_Load_Feed : BOOL;
    HMIPB_RY_S1_Center_VariableSpeedMotor : BOOL;
    RY_S1_Center_VariableSpeedMotor : BOOL;
    SNR_S1_UnLoad_Feed : BOOL;
    LS_S1_UnLoad_UpDownOut : BOOL;
    LS_S1_UnLoad_ConveyorClip1Back : BOOL;
    LS_S1_UnLoad_ConveyorClip2Back : BOOL;
    LS_S1_UnLoad_UpDownBack : BOOL;
    LS_S1_UnLoad_FixClipBack : BOOL;
    HMIPB_YAMAHA_Load_ChangePanelStart : BOOL;
    YAMAHA_ORG : BOOL;
    StepMode : BOOL;
    LS_S1_Load_AlignmentClipBack : BOOL;
    Manual2AutoFlag : BOOL;
    LS_S1_Load_UpDownBack : BOOL;
    LS_S1_Load_ConveyorClip1Back : BOOL;
    LS_S1_Load_ConveyorClip2Back : BOOL;
    LS_S1_Load_FixClipBack : BOOL;
END_VAR
(*
程序名稱: 收盤程序
作者:蔡相偉
版本,日期,版本資訊:
1.0.0		2017/11/16		初始版本

PowerOn=0--->
Idle=1--->
換盤程序開始=2|--->工件取放處無盤=10--->固定,活動,軌道夾持出=11--->上下出=12--->軌道夾持回=13--->上下回=14--->固定夾持回=15--->活動夾持回=16--->換盤完成=17--->1
						  |--->工件取放處有盤=20--->軌道夾持回=21--->固定,活動夾持出=22--->馬達ON=23--->馬達運行中=24--->盤離位,定速馬達停止=25--->10
*)
(*
Error Code
1:緊急停止
2:磁簧異常
*)
//***************************************************************************************************************
//Define
ErrorLS:=
ErrorStatus_S1_FeedPanelUnLoad;
//***************************************************************************************************************
//PowerOn=0
IF NOT(SystemReadyStatus AND NOT(ErrorLS) AND  NOT(Error_PB_EStop)) THEN
	Autoflow:=0;
END_IF;

//Idle=1
IF Autoflow=0 AND SystemReadyStatus AND NOT(ErrorLS) AND  NOT(Error_PB_Estop) THEN
	Autoflow:=1;
END_IF;

IF Autoflow=17 AND NOT(YAMAHA_Unload_ChangePanelStart) AND NOT(HMIPB_YAMAHA_Unload_ChangePanelStart) THEN
	Autoflow:=1;
END_IF;

TON_1(In:=Autoflow=1 AND NOT(SNR_S1_UnLoad_PanelClip), PT:=t#1s);

TON_7(In:=(SNR_S1_UnLoad_PanelClip), PT:=t#1s);
IF Autoflow=1 AND TON_7.Q THEN		(*READY訊號*)
	YAMAHA_UnLoad_Ready:=TRUE;
ELSE
	YAMAHA_UnLoad_Ready:=FALSE;
END_IF;
//換盤程序開始=2
IF Autoflow=1 AND (YAMAHA_Unload_ChangePanelStart OR HMIPB_YAMAHA_Unload_ChangePanelStart) AND NOT(SNR_S1_UnLoad_PanelFeed) THEN
	Autoflow:=2;
END_IF;
IF Autoflow=2 THEN
	HMIPB_RY_S1_Center_VariableSpeedMotor:=TRUE;
END_IF;

//工件取放處無盤=10
IF Autoflow=2 AND NOT(SNR_S1_UnLoad_PanelClip) THEN
	Autoflow:=10;
END_IF;

IF Autoflow=25 THEN
	Autoflow:=10;
END_IF;

//固定,活動,軌道夾持出=11
IF Autoflow=10 THEN
	Autoflow:=11;
END_IF;
TON_8(In:=Autoflow=11 AND NOT(SNR_S1_UnLoad_Feed) AND NOT(StepMode), PT:=t#10s);
IF TON_8.Q THEN
	HMIPB_YAMAHA_Load_ChangePanelStart:=TRUE;
END_IF;
TON_9(In:=HMIPB_YAMAHA_Load_ChangePanelStart, PT:=t#100ms);
//換盤訊號完成=100
IF Autoflow=11 AND TON_9.Q THEN
	Autoflow:=100;
	HMIPB_YAMAHA_Load_ChangePanelStart:=FALSE;
END_IF;
IF Autoflow=11 AND  LS_S1_UnLoad_FixClipOut AND LS_S1_UnLoad_AlignmentClipOut AND LS_S1_UnLoad_ConveyorClip1Out AND LS_S1_UnLoad_ConveyorClip2Out  AND SNR_S1_UnLoad_Feed THEN
	Autoflow:=100;
END_IF;
TON_4(In:=(SNR_S1_UnLoad_Feed), PT:=t#1s);
//上下出=12
IF Autoflow=100 AND LS_S1_UnLoad_FixClipOut AND LS_S1_UnLoad_AlignmentClipOut AND LS_S1_UnLoad_ConveyorClip1Out AND LS_S1_UnLoad_ConveyorClip2Out AND TON_4.Q AND (Rtrig_test.Q OR NOT(StepMode)) THEN
	Autoflow:=12;
	HMIPB_YAMAHA_Load_ChangePanelStart:=FALSE;
END_IF;

//軌道夾持回=13
IF Autoflow=12 AND LS_S1_UnLoad_UpDownOut AND (Rtrig_test.Q OR NOT(StepMode)) THEN
	Autoflow:=13;
END_IF;

//上下回=14
IF Autoflow=13 AND LS_S1_UnLoad_ConveyorClip1Back AND LS_S1_UnLoad_ConveyorClip2Back AND (Rtrig_test.Q OR NOT(StepMode)) THEN
	Autoflow:=14;
END_IF;

//固定夾持回=15
IF Autoflow=14 AND LS_S1_UnLoad_UpDownBack AND (Rtrig_test.Q OR NOT(StepMode)) THEN
	Autoflow:=15;
END_IF;

//活動夾持回=16
IF Autoflow=15 AND LS_S1_UnLoad_FixClipBack AND (Rtrig_test.Q OR NOT(StepMode)) THEN
	Autoflow:=16;
END_IF;

//換盤完成=17
IF Autoflow=16 AND LS_S1_UnLoad_AlignmentClipBack THEN
	Autoflow:=17;
END_IF;

//***************************************************************************************************************
//工件取放處有盤=20
IF Autoflow=2 AND (SNR_S1_UnLoad_PanelClip) THEN
	Autoflow:=20;
END_IF;

//軌道夾持回=21
IF Autoflow=20 THEN
	Autoflow:=21;
END_IF;

//固定,活動夾持出=22
IF Autoflow=21 AND LS_S1_UnLoad_ConveyorClip1Back AND LS_S1_UnLoad_ConveyorClip2Back AND (Rtrig_test.Q OR NOT(StepMode)) THEN
	Autoflow:=22;
END_IF;

//馬達ON=23
IF Autoflow=22 AND YAMAHA_ORG AND LS_S1_UnLoad_FixClipOut AND LS_S1_UnLoad_AlignmentClipOut AND NOT(SNR_S1_UnLoad_PanelFeed) AND (Rtrig_test.Q OR NOT(StepMode)) THEN
	Autoflow:=23;
END_IF;
IF Autoflow=23 THEN
	HMIPB_RY_S1_UnLoad_FixSpeedMotor:=TRUE;
	HMIPB_RY_S1_UnLoad_VariableSpeedMotor:=TRUE;
END_IF;

//馬達運行中=24
IF Autoflow=23 AND RY_S1_UnLoad_FixSpeedMotor AND RY_S1_UnLoad_VariableSpeedMotor THEN
	Autoflow:=24;
END_IF;

//盤離位,定速馬達停止=25
IF Autoflow=24 AND NOT(SNR_S1_UnLoad_PanelClip) AND NOT(RY_S1_UnLoad_FixSpeedMotor) THEN
	Autoflow:=25;
END_IF;

//***************************************************************************************************************
//下夾板出盤固定邊定位電磁閥
R_TRIG_1[0](CLK:=HMIPB_SOL_S1_UnLoad_FixClip AND NOT(AutoStatus));
interlockback[0]:=TRUE;
interlockout[0]:=TRUE;
//SET
IF ((R_TRIG_1[0].Q AND NOT(solStatus[0])) OR Autoflow=11 OR Autoflow=22) AND interlockout[0] THEN
	SOL_S1_UnLoad_FixClip:=TRUE;
END_IF;
//RESET
IF ((R_TRIG_1[0].Q AND (solStatus[0])) OR Autoflow=15 OR Initflow=26) AND interlockback[0] THEN
	SOL_S1_UnLoad_FixClip:=FALSE;
END_IF;
//STATUS
solStatus[0]:=SOL_S1_UnLoad_FixClip;
//***************************************************************************************************************
//下夾板出盤活動邊定位電磁閥
R_TRIG_1[1](CLK:=HMIPB_SOL_S1_UnLoad_AlignmentClip AND NOT(AutoStatus));
interlockback[1]:=TRUE;
interlockout[1]:=TRUE;
//SET
IF ((R_TRIG_1[1].Q AND NOT(solStatus[1])) OR Autoflow=11 OR Autoflow=22) AND interlockout[1] THEN
	SOL_S1_UnLoad_AlignmentClip:=TRUE;
END_IF;
//RESET
IF ((R_TRIG_1[1].Q AND (solStatus[1])) OR Autoflow=16 OR Initflow=27) AND interlockback[1] THEN
	SOL_S1_UnLoad_AlignmentClip:=FALSE;
END_IF;
//STATUS
solStatus[1]:=SOL_S1_UnLoad_AlignmentClip;
//***************************************************************************************************************
//下夾板出盤軌道開合電磁閥
R_TRIG_1[2](CLK:=HMIPB_SOL_S1_UnLoad_ConveyorClip AND NOT(AutoStatus));
interlockback[2]:=TRUE;
interlockout[2]:=TRUE;
//SET
IF ((R_TRIG_1[2].Q AND NOT(solStatus[2])) OR Autoflow=11) AND interlockout[2] THEN
	SOL_S1_UnLoad_ConveyorClip:=TRUE;
END_IF;
//RESET
IF ((R_TRIG_1[2].Q AND (solStatus[2])) OR Autoflow=13 OR Autoflow=21 OR Initflow=21) AND interlockback[2] THEN
	SOL_S1_UnLoad_ConveyorClip:=FALSE;
END_IF;
//STATUS
solStatus[2]:=SOL_S1_UnLoad_ConveyorClip;
//***************************************************************************************************************
//下夾板出盤升降電磁閥
R_TRIG_1[3](CLK:=HMIPB_SOL_S1_UnLoad_UpDown AND NOT(AutoStatus));
interlockback[3]:=TRUE;
interlockout[3]:=LS_S1_UnLoad_ConveyorClip1Out AND LS_S1_UnLoad_ConveyorClip2Out AND SOL_S1_UnLoad_ConveyorClip;
//SET
IF ((R_TRIG_1[3].Q AND NOT(solStatus[3])) OR Autoflow=12) AND interlockout[3] THEN
	SOL_S1_UnLoad_UpDown:=TRUE;
END_IF;
//RESET
IF ((R_TRIG_1[3].Q AND (solStatus[3])) OR Autoflow=14 OR Initflow=14) AND interlockback[3] THEN
	SOL_S1_UnLoad_UpDown:=FALSE;
END_IF;
//STATUS
solStatus[3]:=SOL_S1_UnLoad_UpDown;
//***************************************************************************************************************
//下夾板出盤調速馬達繼電器
//RESET
TON_6(In:=(SNR_S1_UnLoad_PanelFeed), PT:=t#1s);
IF TON_6.Q THEN
	HMIPB_RY_S1_UnLoad_VariableSpeedMotor:=FALSE;
END_IF;
//OUT
RY_S1_UnLoad_VariableSpeedMotor:=HMIPB_RY_S1_UnLoad_VariableSpeedMotor AND NOT(StepMode);
//***************************************************************************************************************
//下夾板出盤定速馬達繼電器
//RESET
TON_5(In:=NOT(SNR_S1_UnLoad_PanelClip), PT:=t#1s);
IF TON_5.Q THEN
	HMIPB_RY_S1_UnLoad_FixSpeedMotor:=FALSE;
END_IF;
//OUT
RY_S1_UnLoad_FixSpeedMotor:=HMIPB_RY_S1_UnLoad_FixSpeedMotor AND NOT(StepMode);

//***************************************************************************************************************
(*
程序名稱: Feed Panel UnLOAD RESET程序
作者:蔡相偉
版本,日期,版本資訊:
1.0.0		2017/11/16		初始版本

PowerOn=0
Idle=1
上下回=14
軌道夾持回=21
固定邊夾持回=26
活動邊夾持回=27
*)
//***************************************************************************************************************
//PowerOn=0
IF NOT(SystemReadyStatus) THEN
	Initflow:=0;
END_IF;

//Idle=1
IF Initflow=0 AND SystemReadyStatus THEN
	Initflow:=1;
END_IF;

IF Initflow=27 AND LS_S1_UnLoad_AlignmentClipBack THEN
	Initflow:=1;
END_IF;

F_TRIG_1(Clk:=ErrorLS OR Error_PB_Estop);
//上下回=14
IF Initflow=1 AND (F_TRIG_1.Q OR Manual2AutoFlag) THEN
	Initflow:=14;
END_IF;

//軌道夾持回=21
IF Initflow=14 AND LS_S1_UnLoad_UpDownBack THEN
	Initflow:=21;
END_IF;

//固定邊夾持回=26
IF Initflow=21 AND LS_S1_UnLoad_ConveyorClip1Back AND LS_S1_UnLoad_ConveyorClip2Back THEN
	Initflow:=26;
END_IF;

//活動邊夾持回=27
IF Initflow=26 AND LS_S1_UnLoad_FixClipBack THEN
	Initflow:=27;
END_IF;
END_PROGRAM

PROGRAM prStation2
VAR
    interlockback : ARRAY[0..1] OF BOOL;
    interlockout : ARRAY[0..1] OF BOOL;
    solstatus : ARRAY[0..1] OF BOOL;
    R_TRIG_1 : ARRAY[0..1] OF R_TRIG;
    Rtrig_test : R_TRIG;
    F_TRIG_1 : F_TRIG;
    Autoflow : INT;
    Initflow : INT;
    TON1 : TON;
    TON2 : TON;
    TON_CT : TON;
END_VAR
VAR_EXTERNAL
    IndexData : ARRAY[0..19] OF stIndexData;
    DisablePB : ARRAY[0..19] OF BOOL;
    SystemReadyStatus : BOOL;
    AutoStatus : BOOL;
    ErrorStatus : ARRAY[0..19] OF BOOL;
    Error_PB_EStop : BOOL;
    LS_S2_UpDownBack : BOOL;
    MachineRunStatus : BOOL;
    LS_S2_UpDownOut : BOOL;
    HMIPB_SOL_S2_UpDown : BOOL;
    SNR_Index : BOOL;
    RY_Index : BOOL;
    SOL_S2_UpDown : BOOL;
    Manual2AutoFlag : BOOL;
    TestPB : ARRAY[0..19] OF BOOL;
    CycleTime : ARRAY[0..19] OF REAL;
    BatchIndexCount : DINT;
    Error_LS_S2_UpDownOut : BOOL;
    Error_LS_S2_UpDownOut1 : BOOL;
    StepMode : BOOL;
    Error_SNR_S5_Check : BOOL;
    BatchNGCount : DINT;
END_VAR
(*************************************************************************
程序名稱:第2站檢查下夾板流程
作者:蔡相偉
版本,日期,版本資訊:
1.0.0		2017/11/22		初始版本

PowerOn=0
Idle=1
上下出=2
檢查開始=3
上下回=4
*************************************************************************)
(*************************************************************************
異常碼
急停=1
氣缸=2
檢查NG=3
*************************************************************************)
//*************************************************************************
//本站狀態判斷
IF IndexData[2].OKFlag[2]
	OR IndexData[2].NGFlag[2] THEN
	IndexData[2].FinishFlag[2]:=TRUE;
END_IF;
//前站狀態判斷
IF  NOT(IndexData[2].FinishFlag[1]) or	IndexData[2].NGFlag[1] THEN
	IndexData[2].NGFlag[2]:=TRUE;
END_IF;
//本站關閉判斷
IF DisablePB[2] AND IndexData[2].FinishFlag[1] AND IndexData[2].OKFlag[1] AND NOT(IndexData[2].NGFlag[1]) THEN
	IndexData[2].OKFlag[2]:=TRUE;
END_IF;

Rtrig_test(CLK:=TestPB[2]);
//PowerOn=0
IF NOT(SystemReadyStatus AND AutoStatus AND NOT(ErrorStatus[2]) AND NOT(Error_PB_EStop)) THEN
	Autoflow:=0;
END_IF;
	//EStop異常碼
	IF Error_PB_Estop AND NOT(IndexData[2].FinishFlag[2]) AND IndexData[2].OkFlag[1] THEN
		IndexData[2].NGFlag[2]:=TRUE;
		IndexData[2].ErrorLog[2]:=1;
		BatchIndexCount:=BatchIndexCount-1;
		BatchNGCount:=BatchNGCount+1;
	END_IF;
	//Error異常碼
	IF ErrorStatus[2] AND NOT(IndexData[2].FinishFlag[2]) AND IndexData[2].OkFlag[1] THEN
		IndexData[2].NGFlag[2]:=TRUE;
		IndexData[2].ErrorLog[2]:=2;
		BatchIndexCount:=BatchIndexCount-1;
		BatchNGCount:=BatchNGCount+1;
	END_IF;
//Idle=1
IF AutoFlow=0 AND SystemReadyStatus AND AutoStatus AND NOT(ErrorStatus[2]) AND NOT(Error_PB_EStop) THEN
	AutoFlow:=1;
END_IF;

IF Autoflow=4 AND LS_S2_UpDownBack THEN
	Autoflow:=1;
END_IF;

//上下出=2
IF Autoflow=1
	AND AutoStatus
	AND NOT(DisablePB[2])
	AND LS_S2_UpDownBack
	AND NOT(SOL_S2_UpDown)
	AND (MachineRunStatus AND NOT(IndexData[2].FinishFlag[2]) AND IndexData[2].FinishFlag[1] AND IndexData[2].OKFlag[1] AND NOT(IndexData[2].NGFlag[1])
	OR Rtrig_test.Q) THEN
	Autoflow:=2;
	Error_LS_S2_UpDownOut1:=FALSE;
END_IF;

//檢查開始=3
IF Autoflow=2 AND NOT(LS_S2_UpDownBack) THEN
	Autoflow:=3;
END_IF;
TON1(In:=Autoflow=3 AND LS_S2_UpDownOut, PT:=t#500ms);		//OK
TON2(In:=Autoflow=3 AND NOT(TON1.Q), PT:=t#7000ms);		//NG
//上下回=4
IF Autoflow=3 AND TON1.Q AND (Rtrig_test.Q OR NOT(StepMode)) THEN
	IndexData[2].OKFlag[2]:=TRUE;
	IndexData[2].NGFlag[2]:=FALSE;
	IndexData[2].ErrorLog[2]:=0;
	Autoflow:=4;
END_IF;

IF Autoflow=3 AND TON2.Q THEN
	Error_LS_S2_UpDownOut1:=TRUE;
	IndexData[2].OKFlag[2]:=FALSE;
	IndexData[2].NGFlag[2]:=TRUE;
	IndexData[2].ErrorLog[2]:=3;
	BatchIndexCount:=BatchIndexCount-1;
	BatchNGCount:=BatchNGCount+1;
	Autoflow:=4;
END_IF;
//*************************************************************************
//手動
//上下電磁閥
R_TRIG_1[0](CLK:=HMIPB_SOL_S2_UpDown AND NOT(AutoStatus));
interlockback[0]:=TRUE;
interlockout[0]:=SNR_Index AND NOT(RY_Index);
(*SET*)
IF ((R_TRIG_1[0].Q AND NOT(solstatus[0])) OR Autoflow=2) AND interlockout[0] THEN
	SOL_S2_UpDown:=TRUE;
END_IF;
(*RESET*)
IF ((R_TRIG_1[0].Q AND (solstatus[0])) OR Autoflow=4 OR Initflow=4) AND interlockback[0] THEN
	SOL_S2_UpDown:=FALSE;
END_IF;
(*STATUS*)
solstatus[0]:=SOL_S2_UpDown;
(*************************************************************************
程序名稱:第2站檢查下夾板RESET流程
作者:蔡相偉
版本,日期,版本資訊:
1.0.0		2017/11/22		初始版本

PowerOn=0
Idle=1
上下回=4
*************************************************************************)
//PowerOn=0
IF NOT(SystemReadyStatus) THEN
	Initflow:=0;
END_IF;

//Idle=1
IF Initflow=0 AND SystemReadyStatus THEN
	Initflow:=1;
END_IF;

IF Initflow=4 AND LS_S2_UpDownBack THEN
	Initflow:=1;
END_IF;

//上下回=4
F_TRIG_1(CLK:= ErrorStatus[2] OR Error_PB_Estop);
IF Initflow=1 AND (F_TRIG_1.Q OR Manual2AutoFlag) THEN
	Initflow:=4;
END_IF;

//*************************************************************************
//Cycle Time
//*************************************************************************
TON_CT(In:=AutoFlow>1, PT:=t#500s);
IF Autoflow>1 THEN
CycleTime[2]:=LINT_TO_REAL(TimeToNanoSec( TON_CT.ET))/1000000000.0;
END_IF;
END_PROGRAM

PROGRAM prStation4
VAR
    interlockback : ARRAY[0..3] OF BOOL;
    interlockout : ARRAY[0..3] OF BOOL;
    solstatus : ARRAY[0..3] OF BOOL;
    R_TRIG_1 : ARRAY[0..3] OF R_TRIG;
    Rtrig_test : R_TRIG;
    F_TRIG_1 : F_TRIG;
    Autoflow : INT;
    Initflow : INT;
    TON1 : TON;
    TON2 : TON;
    TON_CT : TON;
END_VAR
VAR_EXTERNAL
    HMIPB_SOL_S4_MoveBack : BOOL;
    AutoStatus : BOOL;
    SOL_S4_MoveBack : BOOL;
    SOL_S4_MoveOut : BOOL;
    LS_S4_MoveBack : BOOL;
    HMIPB_SOL_S4_MoveOut : BOOL;
    LS_S4_MoveOut : BOOL;
    HMIPB_SOL_S4_UpDown : BOOL;
    SOL_S4_UpDown : BOOL;
    HMIPB_SOL_S4_Clip : BOOL;
    SOL_S4_Clip : BOOL;
    IndexData : ARRAY[0..19] OF stIndexData;
    DisablePB : ARRAY[0..19] OF BOOL;
    TestPB : ARRAY[0..19] OF BOOL;
    SystemReadyStatus : BOOL;
    ErrorStatus : ARRAY[0..19] OF BOOL;
    Error_PB_EStop : BOOL;
    SOL_S4_THMoveBack : BOOL;
    Error_SNR_S4_Feed : BOOL;
    LS_S4_THMoveBack : BOOL;
    LS_S4_UpDownBack : BOOL;
    LS_S4_ClipBack : BOOL;
    MachineRunStatus : BOOL;
    LS_S4_UpDownOut : BOOL;
    LS_S4_ClipOut : BOOL;
    SNR_Index : BOOL;
    RY_Index : BOOL;
    SOL_S4_THMoveOut : BOOL;
    Manual2AutoFlag : BOOL;
    HMIPB_SOL_S4_THMoveBack : BOOL;
    HMIPB_SOL_S4_THMoveOut : BOOL;
    LS_S4_THMoveOut : BOOL;
    YAMAHA_ORG : BOOL;
    SNR_S4_Feed : BOOL;
    FeedStart : ARRAY[0..19] OF BOOL;
    FeedFinish : ARRAY[0..19] OF BOOL;
    ErrorStatus_TH : ARRAY[0..19] OF BOOL;
    LS_S2_UpDownOut : BOOL;
    CycleTime : ARRAY[0..19] OF REAL;
    BatchIndexCount : DINT;
    Error_LS_S4_UpDownOut1 : BOOL;
    StepMode : BOOL;
    BatchNGCount : DINT;
END_VAR
(*************************************************************************
程序名稱:第4站轉子組流程
作者:蔡相偉
版本,日期,版本資訊:
1.0.0		2017/11/22		初始版本

PowerOn=0
Idle=1
上下出=2
夾取出=3
上下回=4
移位出=5
上下出=6
夾取回=7
上下回=8
移位回=9
*************************************************************************)
(*************************************************************************
異常碼
急停=1
氣缸=2
轉子組放入失敗=3
*************************************************************************)
//*************************************************************************
//本站狀態判斷
IF IndexData[4].OKFlag[4]
	OR IndexData[4].NGFlag[4] THEN
	IndexData[4].FinishFlag[4]:=TRUE;
END_IF;
IF NOT(IndexData[4].FinishFlag[2]) OR 	IndexData[4].NGFlag[2] THEN
	IndexData[4].NGFlag[4]:=TRUE;
END_IF;

IF DisablePB[4] AND IndexData[4].FinishFlag[2] AND IndexData[4].OKFlag[2] AND NOT(IndexData[4].NGFlag[2]) THEN
	IndexData[4].OKFlag[4]:=TRUE;
END_IF;

Rtrig_test(CLK:=TestPB[4]);
//PowerOn=0
IF NOT(SystemReadyStatus AND AutoStatus AND NOT(ErrorStatus[4]) AND NOT(Error_PB_EStop)) THEN
	Autoflow:=0;
END_IF;
	//EStop異常碼
	IF Error_PB_Estop AND NOT(IndexData[4].FinishFlag[4]) AND IndexData[4].OkFlag[1] THEN
		IndexData[4].NGFlag[4]:=TRUE;
		IndexData[4].ErrorLog[4]:=1;
		BatchIndexCount:=BatchIndexCount-1;
		BatchNGCount:=BatchNGCount+1;
	END_IF;
	//Error異常碼
	IF ErrorStatus[4] AND NOT(IndexData[4].FinishFlag[4]) AND IndexData[4].OkFlag[1] THEN
		IndexData[4].NGFlag[4]:=TRUE;
		IndexData[4].ErrorLog[4]:=2;
		BatchIndexCount:=BatchIndexCount-1;
		BatchNGCount:=BatchNGCount+1;
	END_IF;
//Idle=1
IF AutoFlow=0 AND SystemReadyStatus AND AutoStatus AND NOT(ErrorStatus[4]) AND NOT(Error_PB_EStop) THEN
	AutoFlow:=1;
END_IF;

IF Autoflow=9 AND LS_S4_MoveBack THEN
	Autoflow:=1;
END_IF;

//上下出=2
IF Autoflow=1
	AND AutoStatus
	AND NOT(DisablePB[4])
	AND LS_S4_THMoveBack
	AND LS_S4_MoveBack
	AND LS_S4_UpDownBack
	AND LS_S4_ClipBack
	AND SNR_S4_Feed
	AND (MachineRunStatus AND NOT(IndexData[4].FinishFlag[4]) AND IndexData[4].FinishFlag[2] AND IndexData[4].OKFlag[2] AND NOT(IndexData[4].NGFlag[2])
	OR Rtrig_test.Q) THEN
	Autoflow:=2;
	Error_LS_S4_UpDownOut1:=FALSE;
END_IF;

//夾取出=3
IF Autoflow=2 AND LS_S4_UpDownOut AND (Rtrig_test.Q OR NOT(StepMode)) THEN
	Autoflow:=3;
END_IF;

//上下回=4
IF Autoflow=3 AND LS_S4_ClipOut AND (Rtrig_test.Q OR NOT(StepMode)) THEN
	Autoflow:=4;
END_IF;

//移位出=5
IF Autoflow=4 AND LS_S4_UpDownBack AND (Rtrig_test.Q OR NOT(StepMode)) THEN
	Autoflow:=5;
END_IF;

//上下出=6
IF Autoflow=5 AND LS_S4_MoveOut AND (Rtrig_test.Q OR NOT(StepMode)) THEN
	Autoflow:=6;
END_IF;
TON1(In:=Autoflow=6 AND LS_S4_UpDownOut, PT:=t#500ms);		//OK
TON2(In:=Autoflow=6 AND NOT(TON1.Q), PT:=t#2000ms);		//NG

//夾取回=7
IF Autoflow=6 AND TON1.Q AND (Rtrig_test.Q OR NOT(StepMode)) THEN
	IndexData[4].OKFlag[4]:=TRUE;
	IndexData[4].NGFlag[4]:=FALSE;
	IndexData[4].ErrorLog[4]:=0;
	Autoflow:=7;
END_IF;
IF Autoflow=6 AND TON2.Q AND (Rtrig_test.Q OR NOT(StepMode)) THEN
	Error_LS_S4_UpDownOut1:=TRUE;
	IndexData[4].OKFlag[4]:=FALSE;
	IndexData[4].NGFlag[4]:=TRUE;
	IndexData[4].ErrorLog[4]:=3;
	BatchIndexCount:=BatchIndexCount-1;
	BatchNGCount:=BatchNGCount+1;
	Autoflow:=7;
END_IF;

//上下回=8
IF Autoflow=7 AND LS_S4_ClipBack AND (Rtrig_test.Q OR NOT(StepMode)) THEN
	Autoflow:=8;
END_IF;

//移位回=9
IF Autoflow=8 AND LS_S4_UpDownBack AND (Rtrig_test.Q OR NOT(StepMode)) THEN
	Autoflow:=9;
END_IF;
//*************************************************************************
//手動
//移位歸電磁閥
interlockback[0]:=LS_S4_UpDownBack AND NOT(SOL_S4_UpDown);
IF ((HMIPB_SOL_S4_MoveBack AND NOT(AutoStatus)) OR Autoflow=9 OR Initflow=9) AND interlockback[0] THEN
	SOL_S4_MoveBack:=TRUE;
	SOL_S4_MoveOut:=FALSE;
END_IF;
IF LS_S4_MoveBack THEN
	SOL_S4_MoveBack:=FALSE;
END_IF;

//移位出電磁閥
interlockout[0]:=LS_S4_UpDownBack AND NOT(SOL_S4_UpDown);
IF ((HMIPB_SOL_S4_MoveOut AND NOT(AutoStatus)) OR Autoflow=5) AND interlockout[0] THEN
	SOL_S4_MoveBack:=FALSE;
	SOL_S4_MoveOut:=TRUE;
END_IF;
IF LS_S4_MoveOut THEN
	SOL_S4_MoveOut:=FALSE;
END_IF;

//上下電磁閥
R_TRIG_1[1](CLK:=HMIPB_SOL_S4_UpDown AND NOT(AutoStatus));
interlockback[1]:=TRUE;
interlockout[1]:=((LS_S4_MoveBack AND LS_S4_THMoveBack AND NOT(SOL_S4_THMoveBack) AND NOT(SOL_S4_THMoveOut)) OR
	(LS_S4_MoveOut AND SNR_Index AND NOT(RY_Index))) AND
	NOT(SOL_S4_MoveBack) AND NOT(SOL_S4_MoveOut);
(*SET*)
IF ((R_TRIG_1[1].Q AND NOT(solstatus[1])) OR Autoflow=2 OR Autoflow=6) AND interlockout[1] THEN
	SOL_S4_UpDown:=TRUE;
END_IF;
(*RESET*)
IF ((R_TRIG_1[1].Q AND (solstatus[1])) OR Autoflow=4 OR Autoflow=8 OR Initflow=8) AND interlockback[1] THEN
	SOL_S4_UpDown:=FALSE;
END_IF;
(*STATUS*)
solstatus[1]:=SOL_S4_UpDown;

//夾持電磁閥
R_TRIG_1[2](CLK:=HMIPB_SOL_S4_Clip AND NOT(AutoStatus));
interlockback[2]:=TRUE;
interlockout[2]:=TRUE;
(*SET*)
IF ((R_TRIG_1[2].Q AND NOT(solstatus[2])) OR Autoflow=3) AND interlockout[2] THEN
	SOL_S4_Clip:=TRUE;
END_IF;
(*RESET*)
IF ((R_TRIG_1[2].Q AND (solstatus[2])) OR Autoflow=7 OR Initflow=7) AND interlockback[2] THEN
	SOL_S4_Clip:=FALSE;
END_IF;
(*STATUS*)
solstatus[2]:=SOL_S4_Clip;
(*************************************************************************
程序名稱:第4站轉子組RESET流程
作者:蔡相偉
版本,日期,版本資訊:
1.0.0		2017/11/22		初始版本

PowerOn=0
Idle=1
夾取回=7
上下回=8
移位回=9
*************************************************************************)
//PowerOn=0
IF NOT(SystemReadyStatus) THEN
	Initflow:=0;
END_IF;

//Idle=1
IF Initflow=0 AND SystemReadyStatus THEN
	Initflow:=1;
END_IF;

IF Initflow=9 AND LS_S4_MoveBack THEN
	Initflow:=1;
END_IF;

//夾取回=7
F_TRIG_1(CLK:= ErrorStatus[4] OR Error_PB_Estop);
IF Initflow=1 AND (F_TRIG_1.Q OR Manual2AutoFlag) THEN
	Initflow:=7;
END_IF;

//上下回=8
IF Initflow=7 AND LS_S4_ClipBack THEN
	Initflow:=8;
END_IF;

//移位回=9
IF Initflow=8 AND LS_S4_UpDownBack THEN
	Initflow:=9;
END_IF;

//*************************************************************************
//Cycle Time
//*************************************************************************
TON_CT(In:=AutoFlow>1, PT:=t#500s);
IF Autoflow>1 THEN
CycleTime[4]:=LINT_TO_REAL(TimeToNanoSec( TON_CT.ET))/1000000000.0;
END_IF;
END_PROGRAM

PROGRAM prStation4_TH
VAR
    interlockback : ARRAY[0..1] OF BOOL;
    interlockout : ARRAY[0..1] OF BOOL;
    Autoflow : INT;
    Initflow : INT;
    TON1 : TON;
    TON2 : TON;
    TON3 : TON;
    TON4 : TON;
    Rtrig_test : R_TRIG;
    ServoORG : BOOL;
END_VAR
VAR_EXTERNAL
    LS_S4_UpDownBack : BOOL;
    SOL_S4_UpDown : BOOL;
    LS_S4_MoveBack : BOOL;
    YAMAHA_ORG : BOOL;
    HMIPB_SOL_S4_THMoveBack : BOOL;
    AutoStatus : BOOL;
    SOL_S4_THMoveBack : BOOL;
    SOL_S4_THMoveOut : BOOL;
    LS_S4_THMoveBack : BOOL;
    HMIPB_SOL_S4_THMoveOut : BOOL;
    LS_S4_THMoveOut : BOOL;
    SystemReadyStatus : BOOL;
    ErrorStatus : ARRAY[0..19] OF BOOL;
    Error_PB_EStop : BOOL;
    IndexData : ARRAY[0..19] OF stIndexData;
    ErrorStatus_TH : ARRAY[0..19] OF BOOL;
    SNR_S4_Feed : BOOL;
    FeedStart : ARRAY[0..19] OF BOOL;
    FeedFinish : ARRAY[0..19] OF BOOL;
    Error_SNR_S4_Feed : BOOL;
    PB_Reset : BOOL;
    StepMode : BOOL;
    LS_S4_Center_UpDownBack : BOOL;
    SOL_S4_Center_UpDown : BOOL;
    Ax_Y : stAxis;
    ServoS4_StandbyPosition : LREAL;
    ErrorStatus_S4_Center : BOOL;
    HMIPB_PB_Reset : BOOL;
    Manual2AutoFlag : BOOL;
END_VAR
(*************************************************************************
程序名稱:第4站轉子組節流流程
作者:蔡相偉
版本,日期,版本資訊:
1.0.0		2017/11/22		初始版本

PowerOn=0
Idle=1
無料節流出=2
送料開始=3
送料中=4
送料完成=5
節流回=6
檢查有無料=7
*************************************************************************)
//define
ServoORG:=Ax_Y.lrCurrentPosition>=ServoS4_StandbyPosition-1;

//PowerOn=0
IF NOT(SystemReadyStatus AND AutoStatus AND NOT(ErrorStatus_TH[4]) AND NOT(Error_PB_EStop)) THEN
	Autoflow:=0;
END_IF;

//Idle=1
IF AutoFlow=0 AND SystemReadyStatus AND AutoStatus AND NOT(ErrorStatus[4]) AND NOT(Error_PB_EStop) THEN
	AutoFlow:=1;
END_IF;

IF Autoflow=7 AND (TON2.Q OR TON3.Q) THEN
	Autoflow:=1;
END_IF;

//無料節流出=2
TON1(In:=Autoflow=1 AND LS_S4_THMoveBack AND NOT(SNR_S4_Feed), PT:=t#1s);
IF AutoFlow=1 AND TON1.Q AND NOT(Error_SNR_S4_Feed) THEN
	AutoFlow:=2;
END_IF;

//送料開始=3
IF Autoflow=2 AND LS_S4_THMoveOut THEN
	Autoflow:=3;
END_IF;
IF Autoflow=3 THEN
	FeedStart[4]:=TRUE;
END_IF;
IF FeedFinish[4] OR ErrorStatus_S4_Center THEN
	FeedStart[4]:=FALSE;
END_IF;

//送料中=4
IF Autoflow=3 AND FeedStart[4] THEN
	Autoflow:=4;
END_IF;
TON4(In:=Autoflow=4, PT:=t#12s);
IF TON4.Q THEN
	Error_SNR_S4_Feed:=TRUE;
END_IF;
//送料完成=5
IF Autoflow=4 AND NOT(FeedStart[4]) THEN
	Autoflow:=5;
END_IF;

//節流回=6
IF Autoflow=5 AND (Rtrig_test.Q OR NOT(StepMode)) THEN
	Autoflow:=6;
END_IF;

//檢查有無料=7
IF Autoflow=6 AND LS_S4_THMoveBack THEN
	Autoflow:=7;
END_IF;
TON2(In:=Autoflow=7 AND (SNR_S4_Feed), PT:=t#300ms); 			//OK
TON3(In:=Autoflow=7 AND NOT(SNR_S4_Feed), PT:=t#300ms);	//NG
IF TON3.Q THEN
	Error_SNR_S4_Feed:=TRUE;
END_IF;
IF PB_Reset OR HMIPB_PB_Reset THEN
	Error_SNR_S4_Feed:=FALSE;
END_IF;

//*************************************************************************
//手動
//節流移位歸電磁閥
interlockback[0]:=((LS_S4_UpDownBack AND NOT(SOL_S4_UpDown)) OR NOT(LS_S4_MoveBack)) AND
(LS_S4_Center_UpDownBack AND NOT(SOL_S4_Center_UpDown) OR ServoORG);
IF ((HMIPB_SOL_S4_THMoveBack AND NOT(AutoStatus)) OR Autoflow=6 OR ErrorStatus_TH[4] OR Manual2AutoFlag) AND interlockback[0] THEN
	SOL_S4_THMoveBack:=TRUE;
	SOL_S4_THMoveOut:=FALSE;
END_IF;
IF LS_S4_THMoveBack THEN
	SOL_S4_THMoveBack:=FALSE;
END_IF;

//節流移位出電磁閥
interlockout[0]:=((LS_S4_UpDownBack AND NOT(SOL_S4_UpDown)) OR NOT(LS_S4_MoveBack)) AND
(LS_S4_Center_UpDownBack AND NOT(SOL_S4_Center_UpDown) OR ServoORG);
IF ((HMIPB_SOL_S4_THMoveOut AND NOT(AutoStatus)) OR Autoflow=2) AND interlockout[0] THEN
	SOL_S4_THMoveBack:=FALSE;
	SOL_S4_THMoveOut:=TRUE;
END_IF;
IF LS_S4_THMoveOut THEN
	SOL_S4_THMoveOut:=FALSE;
END_IF;
END_PROGRAM

PROGRAM prStation4_PanelLoad
VAR
    Autoflow : INT;
    Initflow : INT;
    interlockback : ARRAY[0..2] OF BOOL;
    interlockout : ARRAY[0..2] OF BOOL;
    solStatus : ARRAY[0..2] OF BOOL;
    R_TRIG_1 : ARRAY[0..2] OF R_TRIG;
    F_TRIG_1 : F_TRIG;
    ErrorLS : BOOL;
    StartFlag : BOOL;
    FinishFlag : BOOL;
    TON_1 : TON;
    TON_2 : TON;
    TON_3 : TON;
    Rtrig_test : R_TRIG;
END_VAR
VAR_EXTERNAL
    HMIPB_SOL_S4_Load_PanelUpDown1Back : BOOL;
    AutoStatus : BOOL;
    SOL_S4_Load_PanelUpDown1Back : BOOL;
    SOL_S4_Load_PanelUpDown1Out : BOOL;
    LS_S4_Load_PanelUpDown1Back : BOOL;
    HMIPB_SOL_S4_Load_PanelUpDown1Out : BOOL;
    LS_S4_Load_PanelUpDown1Out : BOOL;
    HMIPB_SOL_S4_Load_PanelUpDown2Back : BOOL;
    SOL_S4_Load_PanelUpDown2Back : BOOL;
    SOL_S4_Load_PanelUpDown2Out : BOOL;
    LS_S4_Load_PanelUpDown2Back : BOOL;
    HMIPB_SOL_S4_Load_PanelUpDown2Out : BOOL;
    LS_S4_Load_PanelUpDown2Out : BOOL;
    HMIPB_SOL_S4_Load_PanelClip : BOOL;
    SOL_S4_Load_PanelClip : BOOL;
    ErrorStatus_S4_Load : BOOL;
    FeedStart_S4_Load : BOOL;
    SystemReadyStatus : BOOL;
    Error_PB_EStop : BOOL;
    LS_S4_Load_PanelClip1Out : BOOL;
    LS_S4_Load_PanelClip2Out : BOOL;
    LS_S4_Load_PanelClip2Back : BOOL;
    LS_S4_Load_PanelClip1Back : BOOL;
    FeedFinish_S4_Load : BOOL;
    FeedStart : ARRAY[0..19] OF BOOL;
    FeedFinish : ARRAY[0..19] OF BOOL;
    StepMode : BOOL;
    LS_S1_Load_PanelUpDown1Back : BOOL;
    LS_S1_Load_PanelUpDown2Back : BOOL;
    LS_S1_Load_PanelClip1Back : BOOL;
    LS_S1_Load_PanelClip2Back : BOOL;
    Manual2AutoFlag : BOOL;
END_VAR
(*
程序名稱: Panel LOAD程序
作者:蔡相偉
版本,日期,版本資訊:
1.0.0		2017/11/16		初始版本

PowerOn=0
Idle=1
Panel出盤程序開始=10
第1段,第2段出=2
夾持出=3
第2段回=4
夾持回=5
第1段回=6
第1段到回=7
*)
//***************************************************************************************************************
//Define
ErrorLS:=ErrorStatus_S4_Load;
StartFlag:=FeedStart_S4_Load;
FeedFinish_S4_Load:=FinishFlag;
TON_1(In:=FeedStart_S4_Load, PT:=t#100ms);
//PowerOn=0
IF NOT(SystemReadyStatus AND NOT(ErrorLS) AND  NOT(Error_PB_EStop)) THEN
	Autoflow:=0;
END_IF;

//Idle=1
IF AutoFlow=0 AND SystemReadyStatus AND NOT(ErrorLS) AND  NOT(Error_PB_Estop) THEN
	AutoFlow:=1;
END_IF;

IF Autoflow=7 AND NOT(StartFlag) THEN
	Autoflow:=1;
END_IF;

//第1段,第2段出=2
IF Autoflow=1 AND StartFlag THEN
	Autoflow:=2;
END_IF;

//承盤夾持出=3
IF Autoflow=2 AND LS_S4_Load_PanelUpDown1Out AND LS_S4_Load_PanelUpDown2Out AND (Rtrig_test.Q OR NOT(StepMode)) THEN
	Autoflow:=3;
END_IF;
TON_2(In:= Autoflow=3 AND LS_S4_Load_PanelClip1Out AND LS_S4_Load_PanelClip2Out , PT:=t#300ms);

//第2段回=4
IF Autoflow=3 AND TON_2.Q AND (Rtrig_test.Q OR NOT(StepMode)) THEN
	Autoflow:=4;
END_IF;
TON_3(In:=Autoflow=4 AND LS_S4_Load_PanelUpDown2Back, PT:=t#500ms);

//承盤夾持回=5
IF Autoflow=4 AND TON_3.Q AND (Rtrig_test.Q OR NOT(StepMode)) THEN
	Autoflow:=5;
END_IF;

//第1段回=6
IF Autoflow=5 AND  LS_S4_Load_PanelClip1Back AND LS_S4_Load_PanelClip2Back AND (Rtrig_test.Q OR NOT(StepMode)) THEN
	Autoflow:=6;
END_IF;

//第1段到回=7
IF Autoflow=6 AND  LS_S4_Load_PanelUpDown1Back THEN
	Autoflow:=7;
END_IF;
IF Autoflow=7 THEN
	FinishFlag:=TRUE;
ELSE
	FinishFlag:=FALSE;
END_IF;

//***************************************************************************************************************
//出盤下降第1段回電磁閥
interlockback[0]:=TRUE;
IF ((HMIPB_SOL_S4_Load_PanelUpDown1Back AND NOT(AutoStatus)) OR Autoflow=6 OR Initflow=3) AND interlockback[0] THEN
	SOL_S4_Load_PanelUpDown1Back:=TRUE;
	SOL_S4_Load_PanelUpDown1Out:=FALSE;
END_IF;
IF LS_S4_Load_PanelUpDown1Back THEN
	SOL_S4_Load_PanelUpDown1Back:=FALSE;
END_IF;

//下夾板出盤下降第1段出電磁閥
interlockout[0]:=TRUE;
IF ((HMIPB_SOL_S4_Load_PanelUpDown1Out AND NOT(AutoStatus)) OR Autoflow=2) AND interlockout[0] THEN
	SOL_S4_Load_PanelUpDown1Back:=FALSE;
	SOL_S4_Load_PanelUpDown1Out:=TRUE;
END_IF;
IF LS_S4_Load_PanelUpDown1Out THEN
	SOL_S4_Load_PanelUpDown1Out:=FALSE;
END_IF;
//***************************************************************************************************************
//下夾板出盤下降第2段回電磁閥
interlockback[1]:=TRUE;
IF ((HMIPB_SOL_S4_Load_PanelUpDown2Back AND NOT(AutoStatus)) OR Autoflow=4 OR Initflow=3) AND interlockback[1] THEN
	SOL_S4_Load_PanelUpDown2Back:=TRUE;
	SOL_S4_Load_PanelUpDown2Out:=FALSE;
END_IF;
IF LS_S4_Load_PanelUpDown2Back THEN
	SOL_S4_Load_PanelUpDown2Back:=FALSE;
END_IF;

//下夾板出盤下降第2段出電磁閥
interlockout[1]:=LS_S4_Load_PanelUpDown1Out;
IF ((HMIPB_SOL_S4_Load_PanelUpDown2Out AND NOT(AutoStatus)) OR Autoflow=2) AND interlockout[1] THEN
	SOL_S4_Load_PanelUpDown2Back:=FALSE;
	SOL_S4_Load_PanelUpDown2Out:=TRUE;
END_IF;
IF LS_S4_Load_PanelUpDown2Out THEN
	SOL_S4_Load_PanelUpDown2Out:=FALSE;
END_IF;
//***************************************************************************************************************
(*下夾板出盤承載電磁閥*)
R_TRIG_1[2](CLK:=HMIPB_SOL_S4_Load_PanelClip AND NOT(AutoStatus));
interlockback[2]:=TRUE;
interlockout[2]:=LS_S4_Load_PanelUpDown1Out;
(*SET*)
IF ((R_TRIG_1[2].Q AND NOT(solStatus[2])) OR Autoflow=3) AND interlockout[2] THEN
	SOL_S4_Load_PanelClip:=TRUE;
END_IF;
(*RESET*)
IF ((R_TRIG_1[2].Q AND (solStatus[2])) OR Autoflow=5 OR Initflow=2) AND interlockback[2] THEN
	SOL_S4_Load_PanelClip:=FALSE;
END_IF;
(*STATUS*)
solStatus[2]:=SOL_S4_Load_PanelClip;

//***************************************************************************************************************
(*
程序名稱: Panel LOAD RESET程序
作者:蔡相偉
版本,日期,版本資訊:
1.0.0		2017/11/16		初始版本

PowerOn=0
Idle=1
夾持回=2
第1段回,第2段回=3
*)
//***************************************************************************************************************
//PowerOn=0
IF NOT(SystemReadyStatus) THEN
	Initflow:=0;
END_IF;

//Idle=1
IF Initflow=0 AND SystemReadyStatus THEN
	Initflow:=1;
END_IF;

IF Initflow=3 AND LS_S4_Load_PanelUpDown1Back AND LS_S4_Load_PanelUpDown2Back THEN
	Initflow:=1;
END_IF;

F_TRIG_1(Clk:=ErrorLS OR Error_PB_Estop);
//夾持回=2
IF Initflow=1 AND (F_TRIG_1.Q OR Manual2AutoFlag) THEN
	Initflow:=2;
END_IF;

//第1段回,第2段回=3
IF Initflow=2 AND LS_S4_Load_PanelClip1Back AND LS_S4_Load_PanelClip2Back THEN
	Initflow:=3;
END_IF;
END_PROGRAM

PROGRAM prStation4_PanelUnLoad
VAR
    Autoflow : INT;
    Initflow : INT;
    interlockback : ARRAY[0..2] OF BOOL;
    interlockout : ARRAY[0..2] OF BOOL;
    solStatus : ARRAY[0..2] OF BOOL;
    R_TRIG_1 : ARRAY[0..2] OF R_TRIG;
    F_TRIG_1 : F_TRIG;
    ErrorLS : BOOL;
    StartFlag : BOOL;
    TON_1 : TON;
    FinishFlag : BOOL;
    Rtrig_test : R_TRIG;
END_VAR
VAR_EXTERNAL
    AutoStatus : BOOL;
    SystemReadyStatus : BOOL;
    Error_PB_EStop : BOOL;
    HMIPB_SOL_S4_UnLoad_PanelUpDown1Back : BOOL;
    SOL_S4_UnLoad_PanelUpDown1Back : BOOL;
    SOL_S4_UnLoad_PanelUpDown1Out : BOOL;
    LS_S4_UnLoad_PanelUpDown1Back : BOOL;
    HMIPB_SOL_S4_UnLoad_PanelUpDown1Out : BOOL;
    LS_S4_UnLoad_PanelUpDown1Out : BOOL;
    HMIPB_SOL_S4_UnLoad_PanelUpDown2Back : BOOL;
    LS_S4_UnLoad_PanelUpDown2Back : BOOL;
    SOL_S4_UnLoad_PanelUpDown2Back : BOOL;
    SOL_S4_UnLoad_PanelUpDown2Out : BOOL;
    LS_S4_UnLoad_PanelClip1Out : BOOL;
    LS_S4_UnLoad_PanelClip2Out : BOOL;
    SOL_S4_UnLoad_PanelClip : BOOL;
    HMIPB_SOL_S4_UnLoad_PanelUpDown2Out : BOOL;
    LS_S4_UnLoad_PanelUpDown2Out : BOOL;
    HMIPB_SOL_S4_UnLoad_PanelClip : BOOL;
    FeedFinish_S4_UnLoad : BOOL;
    FeedStart_S4_UnLoad : BOOL;
    ErrorStatus_S4_UnLoad : BOOL;
    LS_S4_UnLoad_PanelClip1Back : BOOL;
    LS_S4_UnLoad_PanelClip2Back : BOOL;
    StepMode : BOOL;
    LS_S1_Load_PanelUpDown1Back : BOOL;
    LS_S1_Load_PanelUpDown2Back : BOOL;
    LS_S1_Load_PanelClip1Back : BOOL;
    LS_S1_Load_PanelClip2Back : BOOL;
    Manual2AutoFlag : BOOL;
END_VAR
(*
程序名稱: Panel UNLOAD程序
作者:蔡相偉
版本,日期,版本資訊:
1.0.0		2017/11/16		初始版本

PowerOn=0
Idle=1
Panel出盤程序開始=10
第1段出=2
夾持出=3
第2段出=4
夾持回=5
第1段,第2段回=6
第1段,第2段到回=7
*)
//***************************************************************************************************************
//Define
ErrorLS:=ErrorStatus_S4_UnLoad;
StartFlag:=FeedStart_S4_UnLoad;
FeedFinish_S4_UnLoad:=FinishFlag;
TON_1(In:=FeedStart_S4_UnLoad, PT:=t#100ms);
//PowerOn=0
IF NOT(SystemReadyStatus AND NOT(ErrorLS) AND  NOT(Error_PB_EStop)) THEN
	Autoflow:=0;
END_IF;

//Idle=1
IF AutoFlow=0 AND SystemReadyStatus AND NOT(ErrorLS) AND  NOT(Error_PB_Estop) THEN
	AutoFlow:=1;
END_IF;

IF Autoflow=7 AND NOT(StartFlag) THEN
	Autoflow:=1;
END_IF;

//第1段出=2
IF Autoflow=1 AND StartFlag THEN
	Autoflow:=2;
END_IF;

//承盤夾持出=3
IF Autoflow=2 AND LS_S4_UnLoad_PanelUpDown1Out AND (Rtrig_test.Q OR NOT(StepMode)) THEN
	Autoflow:=3;
END_IF;

//第2段出=4
IF Autoflow=3 AND LS_S4_UnLoad_PanelClip1Out AND LS_S4_UnLoad_PanelClip2Out AND (Rtrig_test.Q OR NOT(StepMode)) THEN
	Autoflow:=4;
END_IF;

//承盤夾持回=5
IF Autoflow=4 AND LS_S4_UnLoad_PanelUpDown2Out AND (Rtrig_test.Q OR NOT(StepMode)) THEN
	Autoflow:=5;
END_IF;

//第1段,第2段回=6
IF Autoflow=5 AND  LS_S4_UnLoad_PanelClip1Back AND LS_S4_UnLoad_PanelClip2Back AND (Rtrig_test.Q OR NOT(StepMode)) THEN
	Autoflow:=6;
END_IF;

//第1段,第2段到回=7
IF Autoflow=6 AND LS_S4_UnLoad_PanelUpDown1Back AND LS_S4_UnLoad_PanelUpDown2Back THEN
	Autoflow:=7;
END_IF;
IF Autoflow=7 THEN
	FinishFlag:=TRUE;
ELSE
	FinishFlag:=FALSE;
END_IF;
//***************************************************************************************************************
//出盤下降第1段回電磁閥
interlockback[0]:=TRUE;
IF ((HMIPB_SOL_S4_UnLoad_PanelUpDown1Back AND NOT(AutoStatus)) OR Autoflow=6 OR Initflow=3) AND interlockback[0] THEN
	SOL_S4_UnLoad_PanelUpDown1Back:=TRUE;
	SOL_S4_UnLoad_PanelUpDown1Out:=FALSE;
END_IF;
IF LS_S4_UnLoad_PanelUpDown1Back THEN
	SOL_S4_UnLoad_PanelUpDown1Back:=FALSE;
END_IF;

//下夾板出盤下降第1段出電磁閥
interlockout[0]:=TRUE;
IF ((HMIPB_SOL_S4_UnLoad_PanelUpDown1Out AND NOT(AutoStatus)) OR Autoflow=2) AND interlockout[0] THEN
	SOL_S4_UnLoad_PanelUpDown1Back:=FALSE;
	SOL_S4_UnLoad_PanelUpDown1Out:=TRUE;
END_IF;
IF LS_S4_UnLoad_PanelUpDown1Out THEN
	SOL_S4_UnLoad_PanelUpDown1Out:=FALSE;
END_IF;
//***************************************************************************************************************
//下夾板出盤下降第2段回電磁閥
interlockback[1]:=TRUE;
IF ((HMIPB_SOL_S4_UnLoad_PanelUpDown2Back AND NOT(AutoStatus)) OR Autoflow=6 OR Initflow=3) AND interlockback[1] THEN
	SOL_S4_UnLoad_PanelUpDown2Back:=TRUE;
	SOL_S4_UnLoad_PanelUpDown2Out:=FALSE;
END_IF;
IF LS_S4_UnLoad_PanelUpDown2Back THEN
	SOL_S4_UnLoad_PanelUpDown2Back:=FALSE;
END_IF;

//下夾板出盤下降第2段出電磁閥
interlockout[1]:=LS_S4_UnLoad_PanelClip1Out AND LS_S4_UnLoad_PanelClip2Out AND SOL_S4_UnLoad_PanelClip;
IF ((HMIPB_SOL_S4_UnLoad_PanelUpDown2Out AND NOT(AutoStatus)) OR Autoflow=4) AND interlockout[1] THEN
	SOL_S4_UnLoad_PanelUpDown2Back:=FALSE;
	SOL_S4_UnLoad_PanelUpDown2Out:=TRUE;
END_IF;
IF LS_S4_UnLoad_PanelUpDown2Out THEN
	SOL_S4_UnLoad_PanelUpDown2Out:=FALSE;
END_IF;
//***************************************************************************************************************
(*下夾板出盤承載電磁閥*)
R_TRIG_1[2](CLK:=HMIPB_SOL_S4_UnLoad_PanelClip AND NOT(AutoStatus));
interlockback[2]:=TRUE;
interlockout[2]:=LS_S4_UnLoad_PanelUpDown1Out;
(*SET*)
IF ((R_TRIG_1[2].Q AND NOT(solStatus[2])) OR Autoflow=3) AND interlockout[2] THEN
	SOL_S4_UnLoad_PanelClip:=TRUE;
END_IF;
(*RESET*)
IF ((R_TRIG_1[2].Q AND (solStatus[2])) OR Autoflow=5 OR Initflow=2) AND interlockback[2] THEN
	SOL_S4_UnLoad_PanelClip:=FALSE;
END_IF;
(*STATUS*)
solStatus[2]:=SOL_S4_UnLoad_PanelClip;

//***************************************************************************************************************
(*
程序名稱: Panel UnLOAD RESET程序
作者:蔡相偉
版本,日期,版本資訊:
1.0.0		2017/11/16		初始版本

PowerOn=0
Idle=1
夾持回=2
第1段回,第2段回=3
*)
//***************************************************************************************************************
//PowerOn=0
IF NOT(SystemReadyStatus) THEN
	Initflow:=0;
END_IF;

//Idle=1
IF Initflow=0 AND SystemReadyStatus THEN
	Initflow:=1;
END_IF;

IF Initflow=3 AND LS_S4_UnLoad_PanelUpDown1Back AND LS_S4_UnLoad_PanelUpDown2Back THEN
	Initflow:=1;
END_IF;

F_TRIG_1(Clk:=ErrorLS OR Error_PB_Estop);
//夾持回=2
IF Initflow=1 AND (F_TRIG_1.Q OR Manual2AutoFlag) THEN
	Initflow:=2;
END_IF;

//第1段回,第2段回=3
IF Initflow=2 AND LS_S4_UnLoad_PanelClip1Back AND LS_S4_UnLoad_PanelClip2Back THEN
	Initflow:=3;
END_IF;
END_PROGRAM

PROGRAM prStation5
VAR
    interlockback : ARRAY[0..1] OF BOOL;
    interlockout : ARRAY[0..1] OF BOOL;
    solstatus : ARRAY[0..1] OF BOOL;
    R_TRIG_1 : ARRAY[0..1] OF R_TRIG;
    Rtrig_test : R_TRIG;
    F_TRIG_1 : F_TRIG;
    Autoflow : INT;
    Initflow : INT;
    TON1 : TON;
    TON2 : TON;
    TON_CT : TON;
END_VAR
VAR_EXTERNAL
    IndexData : ARRAY[0..19] OF stIndexData;
    DisablePB : ARRAY[0..19] OF BOOL;
    SystemReadyStatus : BOOL;
    AutoStatus : BOOL;
    ErrorStatus : ARRAY[0..19] OF BOOL;
    Error_PB_EStop : BOOL;
    MachineRunStatus : BOOL;
    SNR_Index : BOOL;
    RY_Index : BOOL;
    Manual2AutoFlag : BOOL;
    TestPB : ARRAY[0..19] OF BOOL;
    SNR_S5_Check : BOOL;
    CycleTime : ARRAY[0..19] OF REAL;
    BatchIndexCount : DINT;
    Error_SNR_S5_Check : BOOL;
    PB_Reset : BOOL;
    HMIPB_PB_Reset : BOOL;
    BatchNGCount : DINT;
END_VAR
(*************************************************************************
程序名稱:第5站檢查轉子組流程
作者:蔡相偉
版本,日期,版本資訊:
1.0.0		2017/11/22		初始版本

PowerOn=0
Idle=1
檢查開始=2
檢查完成=3
*************************************************************************)
(*************************************************************************
異常碼
急停=1
氣缸=2
檢查NG=3
*************************************************************************)
//*************************************************************************
//本站狀態判斷
IF IndexData[5].OKFlag[5]
	OR IndexData[5].NGFlag[5] THEN
	IndexData[5].FinishFlag[5]:=TRUE;
END_IF;
//前站狀態判斷
IF  NOT(IndexData[5].FinishFlag[4]) OR	IndexData[5].NGFlag[4] THEN
	IndexData[5].NGFlag[5]:=TRUE;
END_IF;
//本站關閉判斷
IF DisablePB[5] AND IndexData[5].FinishFlag[4] AND IndexData[5].OKFlag[4] AND NOT(IndexData[5].NGFlag[4]) THEN
	IndexData[5].OKFlag[5]:=TRUE;
END_IF;

Rtrig_test(CLK:=TestPB[5]);
//PowerOn=0
IF NOT(SystemReadyStatus AND AutoStatus AND NOT(ErrorStatus[5]) AND NOT(Error_PB_EStop)) THEN
	Autoflow:=0;
END_IF;
	//EStop異常碼
	(*IF Error_PB_Estop AND NOT(IndexData[4].FinishFlag[4]) AND IndexData[4].OkFlag[1] THEN
		IndexData[4].NGFlag[4]:=TRUE;
		IndexData[4].ErrorLog[4]:=1;
	END_IF;*)
	//Error異常碼
	(*IF ErrorStatus[4] AND NOT(IndexData[4].FinishFlag[4]) AND IndexData[4].OkFlag[1] THEN
		IndexData[4].NGFlag[4]:=TRUE;
		IndexData[4].ErrorLog[4]:=2;
	END_IF;*)
//Idle=1
IF AutoFlow=0 AND SystemReadyStatus AND AutoStatus AND NOT(ErrorStatus[5]) AND NOT(Error_PB_EStop) THEN
	AutoFlow:=1;
END_IF;

IF Autoflow=3 AND IndexData[5].FinishFlag[5] THEN
	Autoflow:=1;
END_IF;

//檢查開始=2
IF Autoflow=1
	AND AutoStatus
	AND NOT(DisablePB[5])
	AND SNR_Index
	AND NOT(RY_Index)
	AND (MachineRunStatus AND NOT(IndexData[5].FinishFlag[5]) AND IndexData[5].FinishFlag[4] AND IndexData[5].OKFlag[4] AND NOT(IndexData[5].NGFlag[4])
	OR Rtrig_test.Q) THEN
	Autoflow:=2;
	Error_SNR_S5_Check:=FALSE;
END_IF;
TON1(In:=Autoflow=2 AND SNR_S5_Check, PT:=t#500ms);		//OK
TON2(In:=Autoflow=2 AND NOT(TON1.Q), PT:=t#1000ms);		//NG
//檢查完成=3
IF Autoflow=2 AND TON1.Q AND NOT(IndexData[5].FinishFlag[5]) THEN
	IndexData[5].OKFlag[5]:=TRUE;
	IndexData[5].NGFlag[5]:=FALSE;
	IndexData[5].ErrorLog[5]:=0;
	Autoflow:=3;
END_IF;
IF Autoflow=2 AND TON2.Q AND NOT(IndexData[5].FinishFlag[5]) THEN
	Error_SNR_S5_Check:=TRUE;
	IndexData[5].OKFlag[5]:=FALSE;
	IndexData[5].NGFlag[5]:=TRUE;
	IndexData[5].ErrorLog[5]:=3;
	BatchIndexCount:=BatchIndexCount-1;
	BatchNGCount:=BatchNGCount+1;
	Autoflow:=3;
END_IF;
IF NOT(SNR_Index) THEN
	Error_SNR_S5_Check:=FALSE;
END_IF;
//*************************************************************************
//Cycle Time
//*************************************************************************
TON_CT(In:=AutoFlow>1, PT:=t#500s);
IF Autoflow>1 THEN
CycleTime[5]:=LINT_TO_REAL(TimeToNanoSec( TON_CT.ET))/1000000000.0;
END_IF;
END_PROGRAM

PROGRAM prStation6
VAR
    interlockback : ARRAY[0..3] OF BOOL;
    interlockout : ARRAY[0..3] OF BOOL;
    solstatus : ARRAY[0..3] OF BOOL;
    R_TRIG_1 : ARRAY[0..3] OF R_TRIG;
    Rtrig_test : R_TRIG;
    F_TRIG_1 : F_TRIG;
    F_TRIG_2 : F_TRIG;
    TON_Break : TON;
    Autoflow : INT;
    Initflow : INT;
    TON1 : TON;
    TON2 : TON;
    TON3 : TON;
    TON_CT : TON;
END_VAR
VAR_EXTERNAL
    HMIPB_SOL_S6_MoveBack : BOOL;
    AutoStatus : BOOL;
    SOL_S6_MoveBack : BOOL;
    SOL_S6_MoveOut : BOOL;
    LS_S6_MoveBack : BOOL;
    HMIPB_SOL_S6_MoveOut : BOOL;
    LS_S6_MoveOut : BOOL;
    HMIPB_SOL_S6_UpDown : BOOL;
    SOL_S6_UpDown : BOOL;
    IndexData : ARRAY[0..19] OF stIndexData;
    DisablePB : ARRAY[0..19] OF BOOL;
    TestPB : ARRAY[0..19] OF BOOL;
    SystemReadyStatus : BOOL;
    ErrorStatus : ARRAY[0..19] OF BOOL;
    Error_PB_EStop : BOOL;
    Error_SNR_S6_Feed : BOOL;
    LS_S6_UpDownBack : BOOL;
    MachineRunStatus : BOOL;
    LS_S6_UpDownOut : BOOL;
    SNR_Index : BOOL;
    RY_Index : BOOL;
    Manual2AutoFlag : BOOL;
    YAMAHA_ORG : BOOL;
    SNR_S6_Feed : BOOL;
    FeedStart : ARRAY[0..19] OF BOOL;
    FeedFinish : ARRAY[0..19] OF BOOL;
    ErrorStatus_TH : ARRAY[0..19] OF BOOL;
    LS_S2_UpDownOut : BOOL;
    LS_S6_THBack : BOOL;
    SOL_S6_Vacuum : BOOL;
    SOL_S6_Break : BOOL;
    SNR_S6_Vacuum : BOOL;
    HMIPB_SOL_S6_Vacuum : BOOL;
    SOL_S6_TH : BOOL;
    CycleTime : ARRAY[0..19] OF REAL;
    BatchIndexCount : DINT;
    Error_LS_S6_UpDownOut : BOOL;
    Error_LS_S6_UpDownOut1 : BOOL;
    StepMode : BOOL;
    BatchNGCount : DINT;
END_VAR
(*************************************************************************
程序名稱:第6站齒輪流程
作者:蔡相偉
版本,日期,版本資訊:
1.0.0		2017/11/28		初始版本

PowerOn=0
Idle=1
上下出=2
夾取出=3
上下回=4
移位出=5
上下出=6
夾取回=7
上下回=8
移位回=9
*************************************************************************)
(*************************************************************************
異常碼
急停=1
氣缸=2
轉子組放入失敗=3
*************************************************************************)
//*************************************************************************
//本站狀態判斷
IF IndexData[6].OKFlag[6]
	OR IndexData[6].NGFlag[6] THEN
	IndexData[6].FinishFlag[6]:=TRUE;
END_IF;
IF  NOT(IndexData[6].FinishFlag[5]) OR	IndexData[6].NGFlag[5] THEN
	IndexData[6].NGFlag[6]:=TRUE;
END_IF;

IF DisablePB[6] AND IndexData[6].FinishFlag[5] AND IndexData[6].OKFlag[5] AND NOT(IndexData[6].NGFlag[5]) THEN
	IndexData[6].OKFlag[6]:=TRUE;
END_IF;

Rtrig_test(CLK:=TestPB[6]);
//PowerOn=0
IF NOT(SystemReadyStatus AND AutoStatus AND NOT(ErrorStatus[6]) AND NOT(Error_PB_EStop)) THEN
	Autoflow:=0;
END_IF;
	//EStop異常碼
	IF Error_PB_Estop AND NOT(IndexData[6].FinishFlag[6]) AND IndexData[6].OkFlag[1] THEN
		IndexData[6].NGFlag[6]:=TRUE;
		IndexData[6].ErrorLog[6]:=1;
		BatchNGCount:=BatchNGCount+1;
	END_IF;
	//Error異常碼
	IF ErrorStatus[6] AND NOT(IndexData[6].FinishFlag[6]) AND IndexData[6].OkFlag[1] THEN
		IndexData[6].NGFlag[6]:=TRUE;
		IndexData[6].ErrorLog[6]:=2;
		BatchNGCount:=BatchNGCount+1;
	END_IF;
//Idle=1
IF AutoFlow=0 AND SystemReadyStatus AND AutoStatus AND NOT(ErrorStatus[6]) AND NOT(Error_PB_EStop) THEN
	AutoFlow:=1;
END_IF;

IF Autoflow=9 AND LS_S6_MoveBack THEN
	Autoflow:=1;
END_IF;

//上下出=2
IF Autoflow=1
	AND AutoStatus
	AND NOT(DisablePB[6])
	AND LS_S6_THBack
	AND NOT(Error_SNR_S6_Feed)
	AND LS_S6_MoveBack
	AND LS_S6_UpDownBack
	AND NOT(SOL_S6_Vacuum)
	AND NOT(SOL_S6_Break)
	AND (MachineRunStatus AND NOT(IndexData[6].FinishFlag[6]) AND IndexData[6].FinishFlag[5] AND IndexData[6].OKFlag[5] AND NOT(IndexData[6].NGFlag[5])
	OR Rtrig_test.Q) THEN
	Autoflow:=2;
	Error_LS_S6_UpDownOut1:=FALSE;
END_IF;

//夾取出=3
IF Autoflow=2 AND LS_S6_UpDownOut AND (Rtrig_test.Q OR NOT(StepMode)) THEN
	Autoflow:=3;
END_IF;
TON3(In:=Autoflow=3 AND NOT(SNR_S6_Vacuum), PT:=t#1000ms);
//上下回=4
IF Autoflow=3 AND (SNR_S6_Vacuum OR TON3.Q) AND (Rtrig_test.Q OR NOT(StepMode)) THEN
	Autoflow:=4;
END_IF;

//移位出=5
IF Autoflow=4 AND LS_S6_UpDownBack AND (Rtrig_test.Q OR NOT(StepMode)) THEN
	FeedStart[6]:=TRUE;
	Autoflow:=5;
END_IF;

IF FeedFinish[6] THEN
	FeedStart[6]:=FALSE;
END_IF;

//上下出=6
IF Autoflow=5 AND LS_S6_MoveOut AND (Rtrig_test.Q OR NOT(StepMode)) THEN
	Autoflow:=6;
END_IF;
TON1(In:=Autoflow=6 AND LS_S6_UpDownOut, PT:=t#500ms);		//OK
TON2(In:=Autoflow=6 AND NOT(TON1.Q), PT:=t#2000ms);		//NG

//夾取回=7
IF Autoflow=6 AND TON1.Q AND (Rtrig_test.Q OR NOT(StepMode)) THEN
	IndexData[6].OKFlag[6]:=TRUE;
	IndexData[6].NGFlag[6]:=FALSE;
	IndexData[6].ErrorLog[6]:=0;
	Autoflow:=7;
END_IF;
IF Autoflow=6 AND TON2.Q AND (Rtrig_test.Q OR NOT(StepMode)) THEN
	Error_LS_S6_UpDownOut1:=TRUE;
	IndexData[6].OKFlag[6]:=FALSE;
	IndexData[6].NGFlag[6]:=TRUE;
	IndexData[6].ErrorLog[6]:=3;
	BatchIndexCount:=BatchIndexCount-1;
	BatchNGCount:=BatchNGCount+1;
	Autoflow:=7;
END_IF;

//上下回=8
IF Autoflow=7 AND NOT(SOL_S6_Vacuum) AND NOT(SNR_S6_Vacuum) AND (Rtrig_test.Q OR NOT(StepMode)) THEN
	Autoflow:=8;
END_IF;

//移位回=9
IF Autoflow=8 AND LS_S6_UpDownBack AND (Rtrig_test.Q OR NOT(StepMode)) THEN
	Autoflow:=9;
END_IF;
//*************************************************************************
//手動
//移位歸電磁閥
interlockback[0]:=LS_S6_UpDownBack AND NOT(SOL_S6_UpDown);
IF ((HMIPB_SOL_S6_MoveBack AND NOT(AutoStatus)) OR Autoflow=9 OR Initflow=9) AND interlockback[0] THEN
	SOL_S6_MoveBack:=TRUE;
	SOL_S6_MoveOut:=FALSE;
END_IF;
IF LS_S6_MoveBack THEN
	SOL_S6_MoveBack:=FALSE;
END_IF;

//移位出電磁閥
interlockout[0]:=LS_S6_UpDownBack AND NOT(SOL_S6_UpDown);
IF ((HMIPB_SOL_S6_MoveOut AND NOT(AutoStatus)) OR Autoflow=5) AND interlockout[0] THEN
	SOL_S6_MoveBack:=FALSE;
	SOL_S6_MoveOut:=TRUE;
END_IF;
IF LS_S6_MoveOut THEN
	SOL_S6_MoveOut:=FALSE;
END_IF;

//上下電磁閥
R_TRIG_1[1](CLK:=HMIPB_SOL_S6_UpDown AND NOT(AutoStatus));
interlockback[1]:=TRUE;
interlockout[1]:=((LS_S6_MoveBack AND LS_S6_THBack AND NOT(SOL_S6_TH)) OR
	(LS_S6_MoveOut AND SNR_Index AND NOT(RY_Index))) AND
	NOT(SOL_S6_MoveBack) AND NOT(SOL_S6_MoveOut);
(*SET*)
IF ((R_TRIG_1[1].Q AND NOT(solstatus[1])) OR Autoflow=2 OR Autoflow=6) AND interlockout[1] THEN
	SOL_S6_UpDown:=TRUE;
END_IF;
(*RESET*)
IF ((R_TRIG_1[1].Q AND (solstatus[1])) OR Autoflow=4 OR Autoflow=8 OR Initflow=8) AND interlockback[1] THEN
	SOL_S6_UpDown:=FALSE;
END_IF;
(*STATUS*)
solstatus[1]:=SOL_S6_UpDown;

//吸取電磁閥
R_TRIG_1[2](CLK:=HMIPB_SOL_S6_Vacuum AND NOT(AutoStatus));
interlockback[2]:=TRUE;
interlockout[2]:=TRUE;
(*SET*)
IF ((R_TRIG_1[2].Q AND NOT(solstatus[2])) OR Autoflow=3) AND interlockout[2] THEN
	SOL_S6_Vacuum:=TRUE;
END_IF;
(*RESET*)
IF ((R_TRIG_1[2].Q AND (solstatus[2])) OR Autoflow=7 OR Initflow=7 OR ErrorStatus[6]) AND interlockback[2] THEN
	SOL_S6_Vacuum:=FALSE;
END_IF;
(*STATUS*)
solstatus[2]:=SOL_S6_Vacuum;

//破壞電磁閥
F_TRIG_2(CLK:=SOL_S6_Vacuum);
interlockback[3]:=TRUE;
interlockout[3]:=TRUE;
(*SET*)
IF ((F_TRIG_2.Q AND NOT(solstatus[3]))) AND interlockout[3] THEN
	SOL_S6_Break:=TRUE;
END_IF;
(*RESET*)
TON_Break(In:=SOL_S6_Break, PT:=t#500ms);
IF ((TON_Break.Q AND (solstatus[3]))) AND interlockback[3] THEN
	SOL_S6_Break:=FALSE;
END_IF;
(*STATUS*)
solstatus[3]:=SOL_S6_Break;
(*************************************************************************
程序名稱:第6站齒輪RESET流程
作者:蔡相偉
版本,日期,版本資訊:
1.0.0		2017/11/22		初始版本

PowerOn=0
Idle=1
夾取回=7
上下回=8
移位回=9
*************************************************************************)
//PowerOn=0
IF NOT(SystemReadyStatus) THEN
	Initflow:=0;
END_IF;

//Idle=1
IF Initflow=0 AND SystemReadyStatus THEN
	Initflow:=1;
END_IF;

IF Initflow=9 AND LS_S6_MoveBack THEN
	Initflow:=1;
END_IF;

//夾取回=7
F_TRIG_1(CLK:= ErrorStatus[6] OR Error_PB_Estop);
IF Initflow=1 AND (F_TRIG_1.Q OR Manual2AutoFlag) THEN
	Initflow:=7;
END_IF;

//上下回=8
IF Initflow=7 AND NOT(SOL_S6_Vacuum) AND NOT(SNR_S6_Vacuum) THEN
	Initflow:=8;
END_IF;

//移位回=9
IF Initflow=8 AND LS_S6_UpDownBack THEN
	Initflow:=9;
END_IF;

//*************************************************************************
//Cycle Time
//*************************************************************************
TON_CT(In:=AutoFlow>1, PT:=t#500s);
IF Autoflow>1 THEN
CycleTime[6]:=LINT_TO_REAL(TimeToNanoSec( TON_CT.ET))/1000000000.0;
END_IF;
END_PROGRAM

PROGRAM prStation7
VAR
    interlockback : ARRAY[0..1] OF BOOL;
    interlockout : ARRAY[0..1] OF BOOL;
    solstatus : ARRAY[0..1] OF BOOL;
    R_TRIG_1 : ARRAY[0..1] OF R_TRIG;
    Rtrig_test : R_TRIG;
    F_TRIG_1 : F_TRIG;
    Autoflow : INT;
    Initflow : INT;
    TON1 : TON;
    TON2 : TON;
    TON_CT : TON;
END_VAR
VAR_EXTERNAL
    IndexData : ARRAY[0..19] OF stIndexData;
    DisablePB : ARRAY[0..19] OF BOOL;
    SystemReadyStatus : BOOL;
    AutoStatus : BOOL;
    ErrorStatus : ARRAY[0..19] OF BOOL;
    Error_PB_EStop : BOOL;
    MachineRunStatus : BOOL;
    SNR_Index : BOOL;
    RY_Index : BOOL;
    Manual2AutoFlag : BOOL;
    TestPB : ARRAY[0..19] OF BOOL;
    SNR_S7_Check : BOOL;
    CycleTime : ARRAY[0..19] OF REAL;
    BatchIndexCount : DINT;
    Error_SNR_S7_Check : BOOL;
    PB_Reset : BOOL;
    HMIPB_PB_Reset : BOOL;
    Error_SNR_S5_Check : BOOL;
    BatchNGCount : DINT;
END_VAR
(*************************************************************************
程序名稱:第7站檢查齒輪流程
作者:蔡相偉
版本,日期,版本資訊:
1.0.0		2017/11/22		初始版本

PowerOn=0
Idle=1
檢查開始=2
檢查完成=3
*************************************************************************)
(*************************************************************************
異常碼
急停=1
氣缸=2
檢查NG=3
*************************************************************************)
//*************************************************************************
//本站狀態判斷
IF IndexData[7].OKFlag[7]
	OR IndexData[7].NGFlag[7] THEN
	IndexData[7].FinishFlag[7]:=TRUE;
END_IF;
//前站狀態判斷
IF  NOT(IndexData[7].FinishFlag[6]) OR	IndexData[7].NGFlag[6] THEN
	IndexData[7].NGFlag[7]:=TRUE;
END_IF;
//本站關閉判斷
IF DisablePB[7] AND IndexData[7].FinishFlag[6] AND IndexData[7].OKFlag[6] AND NOT(IndexData[7].NGFlag[6]) THEN
	IndexData[7].OKFlag[7]:=TRUE;
END_IF;

Rtrig_test(CLK:=TestPB[7]);
//PowerOn=0
IF NOT(SystemReadyStatus AND AutoStatus AND NOT(ErrorStatus[7]) AND NOT(Error_PB_EStop)) THEN
	Autoflow:=0;
END_IF;
	//EStop異常碼
	(*IF Error_PB_Estop AND NOT(IndexData[4].FinishFlag[4]) AND IndexData[4].OkFlag[1] THEN
		IndexData[4].NGFlag[4]:=TRUE;
		IndexData[4].ErrorLog[4]:=1;
	END_IF;*)
	//Error異常碼
	(*IF ErrorStatus[4] AND NOT(IndexData[4].FinishFlag[4]) AND IndexData[4].OkFlag[1] THEN
		IndexData[4].NGFlag[4]:=TRUE;
		IndexData[4].ErrorLog[4]:=2;
	END_IF;*)
//Idle=1
IF AutoFlow=0 AND SystemReadyStatus AND AutoStatus AND NOT(ErrorStatus[7]) AND NOT(Error_PB_EStop) THEN
	AutoFlow:=1;
END_IF;

IF Autoflow=3 AND IndexData[7].FinishFlag[7] THEN
	Autoflow:=1;
END_IF;

//檢查開始=2
IF Autoflow=1
	AND AutoStatus
	AND NOT(DisablePB[7])
	AND SNR_Index
	AND NOT(RY_Index)
	AND (MachineRunStatus AND NOT(IndexData[7].FinishFlag[7]) AND IndexData[7].FinishFlag[6] AND IndexData[7].OKFlag[6] AND NOT(IndexData[7].NGFlag[6])
	OR Rtrig_test.Q) THEN
	Autoflow:=2;
	Error_SNR_S7_Check:=FALSE;
END_IF;
TON1(In:=Autoflow=2 AND SNR_S7_Check, PT:=t#500ms);		//OK
TON2(In:=Autoflow=2 AND NOT(TON1.Q), PT:=t#1000ms);		//NG
//檢查完成=3
IF Autoflow=2 AND TON1.Q THEN
	IndexData[7].OKFlag[7]:=TRUE;
	IndexData[7].NGFlag[7]:=FALSE;
	IndexData[7].ErrorLog[7]:=0;
	Autoflow:=3;
END_IF;
IF Autoflow=2 AND TON2.Q THEN
	Error_SNR_S7_Check:=TRUE;
	IndexData[7].OKFlag[7]:=FALSE;
	IndexData[7].NGFlag[7]:=TRUE;
	IndexData[7].ErrorLog[7]:=3;
	BatchIndexCount:=BatchIndexCount-1;
	BatchNGCount:=BatchNGCount+1;
	Autoflow:=3;
END_IF;
IF NOT(SNR_Index) THEN
	Error_SNR_S7_Check:=FALSE;
END_IF;
//*************************************************************************
//Cycle Time
//*************************************************************************
TON_CT(In:=AutoFlow>1, PT:=t#500s);
IF Autoflow>1 THEN
CycleTime[7]:=LINT_TO_REAL(TimeToNanoSec( TON_CT.ET))/1000000000.0;
END_IF;
END_PROGRAM

PROGRAM prStation8
VAR
    interlockback : ARRAY[0..5] OF BOOL;
    interlockout : ARRAY[0..5] OF BOOL;
    solstatus : ARRAY[0..5] OF BOOL;
    R_TRIG_1 : ARRAY[0..5] OF R_TRIG;
    Rtrig_test : R_TRIG;
    F_TRIG_1 : F_TRIG;
    F_TRIG_2 : F_TRIG;
    F_TRIG_3 : F_TRIG;
    TON_BreakF : TON;
    TON_BreakR : TON;
    Autoflow : INT;
    Initflow : INT;
    TON1 : TON;
    TON2 : TON;
    TON3 : TON;
    TON4 : TON;
    TON_CT : TON;
END_VAR
VAR_EXTERNAL
    HMIPB_SOL_S8_MoveBack : BOOL;
    AutoStatus : BOOL;
    SOL_S8_MoveBack : BOOL;
    SOL_S8_MoveOut : BOOL;
    LS_S8_MoveBack : BOOL;
    HMIPB_SOL_S8_MoveOut : BOOL;
    LS_S8_MoveOut : BOOL;
    HMIPB_SOL_S8_UpDown : BOOL;
    SOL_S8_UpDown : BOOL;
    IndexData : ARRAY[0..19] OF stIndexData;
    DisablePB : ARRAY[0..19] OF BOOL;
    TestPB : ARRAY[0..19] OF BOOL;
    SystemReadyStatus : BOOL;
    ErrorStatus : ARRAY[0..19] OF BOOL;
    Error_PB_EStop : BOOL;
    Error_SNR_S8_Feed : BOOL;
    LS_S8_UpDownBack : BOOL;
    MachineRunStatus : BOOL;
    LS_S8_UpDownOut : BOOL;
    SNR_Index : BOOL;
    RY_Index : BOOL;
    Manual2AutoFlag : BOOL;
    YAMAHA_ORG : BOOL;
    SNR_S8_Feed : BOOL;
    FeedStart : ARRAY[0..19] OF BOOL;
    FeedFinish : ARRAY[0..19] OF BOOL;
    ErrorStatus_TH : ARRAY[0..19] OF BOOL;
    LS_S2_UpDownOut : BOOL;
    LS_S8_THBack : BOOL;
    SOL_S8_TH : BOOL;
    HMIPB_SOL_S8_VacuumF : BOOL;
    SOL_S8_VacuumF : BOOL;
    SOL_S8_BreakF : BOOL;
    HMIPB_SOL_S8_VacuumR : BOOL;
    SOL_S8_VacuumR : BOOL;
    SOL_S8_BreakR : BOOL;
    SNR_S8_VacuumF : BOOL;
    SNR_S8_VacuumR : BOOL;
    SNR_S6_Vacuum : BOOL;
    CCDStartFlag : BOOL;
    CCDFinishFlag : BOOL;
    CCD_Check_NG : BOOL;
    S8_ChangeJigStartFlag : BOOL;
    LS_S8_FixBack : BOOL;
    LS_S8_FixMoveOut : BOOL;
    CycleTime : ARRAY[0..19] OF REAL;
    BatchIndexCount : DINT;
    Error_LS_S8_UpDownOut1 : BOOL;
    StepMode : BOOL;
    BatchNGCount : DINT;
END_VAR
(*************************************************************************
程序名稱:第8站卡子流程
作者:蔡相偉
版本,日期,版本資訊:
1.0.0		2017/11/28		初始版本

PowerOn=0
Idle=1
上下出=2
夾取出=3
上下回=4
CCD檢查開始=20
CCD檢查中=21
CCD檢查完成=22
移位出=5
上下出=6
夾取回=7
上下回=8
移位回,換卡子方向=9
*************************************************************************)
(*************************************************************************
異常碼
急停=1
氣缸=2
轉子組放入失敗=3
*************************************************************************)
//*************************************************************************
//本站狀態判斷
IF IndexData[8].OKFlag[8]
	OR IndexData[8].NGFlag[8] THEN
	IndexData[8].FinishFlag[8]:=TRUE;
END_IF;
IF  NOT(IndexData[8].FinishFlag[7]) OR 	IndexData[8].NGFlag[7] THEN
	IndexData[8].NGFlag[8]:=TRUE;
END_IF;

IF DisablePB[8] AND IndexData[8].FinishFlag[7] AND IndexData[8].OKFlag[7] AND NOT(IndexData[8].NGFlag[7]) THEN
	IndexData[8].OKFlag[8]:=TRUE;
END_IF;

Rtrig_test(CLK:=TestPB[8]);
//PowerOn=0
IF NOT(SystemReadyStatus AND AutoStatus AND NOT(ErrorStatus[8]) AND NOT(Error_PB_EStop)) THEN
	Autoflow:=0;
END_IF;
	//EStop異常碼
	IF Error_PB_Estop AND NOT(IndexData[8].FinishFlag[8]) AND IndexData[8].OkFlag[1] THEN
		IndexData[8].NGFlag[8]:=TRUE;
		IndexData[8].ErrorLog[8]:=1;
		BatchIndexCount:=BatchIndexCount-1;
		BatchNGCount:=BatchNGCount+1;
	END_IF;
	//Error異常碼
	IF ErrorStatus[8] AND NOT(IndexData[8].FinishFlag[8]) AND IndexData[8].OkFlag[1] THEN
		IndexData[8].NGFlag[8]:=TRUE;
		IndexData[8].ErrorLog[8]:=2;
		BatchIndexCount:=BatchIndexCount-1;
		BatchNGCount:=BatchNGCount+1;
	END_IF;
//Idle=1
IF AutoFlow=0 AND SystemReadyStatus AND AutoStatus AND NOT(ErrorStatus[8]) AND NOT(Error_PB_EStop) THEN
	AutoFlow:=1;
END_IF;

IF Autoflow=9 AND LS_S8_MoveBack THEN
	Autoflow:=1;
END_IF;

//上下出=2
IF Autoflow=1
	AND AutoStatus
	AND NOT(DisablePB[8])
	AND LS_S8_THBack
	AND NOT(Error_SNR_S8_Feed)
	AND LS_S8_MoveBack
	AND LS_S8_UpDownBack
	AND NOT(SOL_S8_VacuumF)
	AND NOT(SOL_S8_BreakF)
	AND NOT(SOL_S8_VacuumR)
	AND NOT(SOL_S8_BreakR)
	AND (MachineRunStatus AND NOT(IndexData[8].FinishFlag[8]) AND IndexData[8].FinishFlag[7] AND IndexData[8].OKFlag[7] AND NOT(IndexData[8].NGFlag[7])
	OR Rtrig_test.Q) THEN
	Autoflow:=2;
	Error_LS_S8_UpDownOut1:=FALSE;
END_IF;

//夾取出=3
IF Autoflow=2 AND LS_S8_UpDownOut AND (Rtrig_test.Q OR NOT(StepMode)) THEN
	Autoflow:=3;
END_IF;
TON3(In:=Autoflow=3 AND NOT(SNR_S8_VacuumF) AND NOT(SNR_S8_VacuumR), PT:=t#1000ms);
//上下回=4
IF Autoflow=3 AND (SNR_S8_VacuumF AND SNR_S8_VacuumR OR TON3.Q) AND (Rtrig_test.Q OR NOT(StepMode)) THEN
	Autoflow:=4;
	FeedStart[8]:=TRUE;
END_IF;
IF FeedFinish[8] THEN
	FeedStart[8]:=FALSE;
END_IF;
TON4(In:=Autoflow=4 AND LS_S8_UpDownBack, PT:=t#500ms);

//CCD檢查開始=20
IF Autoflow=4 AND TON4.Q THEN
	CCDStartFlag:=TRUE;
	Autoflow:=20;
END_IF;

//CCD檢查中=21
IF Autoflow=20 AND CCDStartFlag THEN
	Autoflow:=21;
END_IF;

//CCD檢查完成=22
IF Autoflow=21 AND CCDFinishFlag THEN
	CCDStartFlag:=FALSE;
	Autoflow:=22;
END_IF;

//移位出=5
IF Autoflow=22 AND (Rtrig_test.Q OR NOT(StepMode)) THEN
	Autoflow:=5;
END_IF;

//上下出=6
IF Autoflow=5 AND LS_S8_MoveOut AND (Rtrig_test.Q OR NOT(StepMode)) THEN
	Autoflow:=6;
END_IF;
TON1(In:=Autoflow=6 AND LS_S8_UpDownOut, PT:=t#500ms);		//OK
TON2(In:=Autoflow=6 AND NOT(TON1.Q), PT:=t#2000ms);		//NG

//夾取回=7
IF Autoflow=6 AND TON1.Q AND (Rtrig_test.Q OR NOT(StepMode)) THEN
	IndexData[8].OKFlag[8]:=TRUE;
	IndexData[8].NGFlag[8]:=FALSE;
	IndexData[8].ErrorLog[8]:=0;
	Autoflow:=7;
END_IF;
IF Autoflow=6 AND TON2.Q AND (Rtrig_test.Q OR NOT(StepMode)) THEN
	Error_LS_S8_UpDownOut1:=TRUE;
	IndexData[8].OKFlag[8]:=FALSE;
	IndexData[8].NGFlag[8]:=TRUE;
	IndexData[8].ErrorLog[8]:=3;
	BatchIndexCount:=BatchIndexCount-1;
	BatchNGCount:=BatchNGCount+1;
	Autoflow:=7;
END_IF;

//上下回=8
IF Autoflow=7 AND NOT(SOL_S8_VacuumF) AND NOT(SNR_S8_VacuumF) AND NOT(SOL_S8_VacuumR) AND NOT(SNR_S8_VacuumR) AND (Rtrig_test.Q OR NOT(StepMode)) THEN
	Autoflow:=8;
END_IF;

//移位回,切換方向=9
IF Autoflow=8 AND LS_S8_UpDownBack AND (Rtrig_test.Q OR NOT(StepMode)) THEN
	IF CCD_Check_NG THEN
		S8_ChangeJigStartFlag:=TRUE;
	END_IF;
	Autoflow:=9;
END_IF;
//*************************************************************************
//手動
//移位歸電磁閥
interlockback[0]:=LS_S8_UpDownBack AND NOT(SOL_S8_UpDown);
IF ((HMIPB_SOL_S8_MoveBack AND NOT(AutoStatus)) OR Autoflow=9 OR Initflow=9) AND interlockback[0] THEN
	SOL_S8_MoveBack:=TRUE;
	SOL_S8_MoveOut:=FALSE;
END_IF;
IF LS_S8_MoveBack THEN
	SOL_S8_MoveBack:=FALSE;
END_IF;

//移位出電磁閥
interlockout[0]:=LS_S8_UpDownBack AND NOT(SOL_S8_UpDown);
IF ((HMIPB_SOL_S8_MoveOut AND NOT(AutoStatus)) OR Autoflow=5) AND interlockout[0] THEN
	SOL_S8_MoveBack:=FALSE;
	SOL_S8_MoveOut:=TRUE;
END_IF;
IF LS_S8_MoveOut THEN
	SOL_S8_MoveOut:=FALSE;
END_IF;

//上下電磁閥
R_TRIG_1[1](CLK:=HMIPB_SOL_S8_UpDown AND NOT(AutoStatus));
interlockback[1]:=TRUE;
interlockout[1]:=((LS_S8_MoveBack AND LS_S8_THBack AND NOT(SOL_S8_TH)) OR
	(LS_S8_MoveOut AND SNR_Index AND NOT(RY_Index))) AND
	NOT(SOL_S8_MoveBack) AND NOT(SOL_S8_MoveOut);
(*SET*)
IF ((R_TRIG_1[1].Q AND NOT(solstatus[1])) OR Autoflow=2 OR Autoflow=6) AND interlockout[1] THEN
	SOL_S8_UpDown:=TRUE;
END_IF;
(*RESET*)
IF ((R_TRIG_1[1].Q AND (solstatus[1])) OR Autoflow=4 OR Autoflow=8 OR Initflow=8) AND interlockback[1] THEN
	SOL_S8_UpDown:=FALSE;
END_IF;
(*STATUS*)
solstatus[1]:=SOL_S8_UpDown;

//前吸取電磁閥
R_TRIG_1[2](CLK:=HMIPB_SOL_S8_VacuumF AND NOT(AutoStatus));
interlockback[2]:=TRUE;
interlockout[2]:=TRUE;
(*SET*)
IF ((R_TRIG_1[2].Q AND NOT(solstatus[2])) OR Autoflow=3) AND interlockout[2] THEN
	SOL_S8_VacuumF:=TRUE;
END_IF;
(*RESET*)
IF ((R_TRIG_1[2].Q AND (solstatus[2])) OR Autoflow=7 OR Initflow=7 OR ErrorStatus[8]) AND interlockback[2] THEN
	SOL_S8_VacuumF:=FALSE;
END_IF;
(*STATUS*)
solstatus[2]:=SOL_S8_VacuumF;

